// TIA Portal V20 export
FUNCTION_BLOCK "Sequence_1_Conveyor"   // FB157, LAD
TITLE = Sequence
// Sequence template programmend in ladder logic
// stored: IsIECCheckEnabled true, MemoryReserve 100, Namespace Unit1.Em7, SetENOAutomatically true
   VAR_INPUT
      UnitStatus : "LAF_typeUnitStatus";
   END_VAR
   VAR_OUTPUT
      safeState : Bool;
   END_VAR
   VAR
      instSequenceLADControl { ExternalWritable := 'False'} : "LAF_ControlLadSequence";
      instSequenceLADStatus { ExternalWritable := 'False'} : "LAF_StatusLadSequence";
      statPulse { ExternalWritable := 'False'} : Array[0..999] of Bool;
      statTonTimer { ExternalWritable := 'False'} : Array[0..1999] of TON_TIME;
   END_VAR
   VAR_TEMP
      tempCustomerAction : Bool;   // Placeholder for possible actions
      tempDo_nothing_and_wait_for_init : Bool;   // Placeholder for doing nothing
      tempSafeStateCondition : Bool;   // Temp Condition for the equipment module to be in a safe state
   END_VAR
   VAR CONSTANT
      STEP_IDLE : DInt := 1;   // Idle Step
      JOB_1_STEP_01 : DInt := 101;
      JOB_1_STEP_11 : DInt := 111;
      JOB_1_STEP_21 : DInt := 121;
      JOB_1_STEP_31 : DInt := 131;
      JOB_1_STEP_41 : DInt := 141;
      JOB_1_STEP_51 : DInt := 151;
      JOB_1_STEP_61 : DInt := 161;
      JOB_1_STEP_71 : DInt := 171;
      JOB_1_STEP_81 : DInt := 181;
      JOB_1_STEP_91 : DInt := 191;
      JOB_2_STEP_01 : DInt := 201;
      JOB_2_STEP_11 : DInt := 211;
      JOB_2_STEP_21 : DInt := 221;
      JOB_2_STEP_31 : DInt := 231;
      JOB_2_STEP_41 : DInt := 241;
      JOB_2_STEP_51 : DInt := 251;
      JOB_2_STEP_61 : DInt := 261;
      JOB_2_STEP_71 : DInt := 271;
      JOB_2_STEP_81 : DInt := 281;
      JOB_2_STEP_91 : DInt := 291;
      JOB_3_STEP_01 : DInt := 301;
      JOB_3_STEP_11 : DInt := 311;
      JOB_3_STEP_21 : DInt := 321;
      JOB_3_STEP_31 : DInt := 331;
      JOB_3_STEP_41 : DInt := 341;
      JOB_3_STEP_51 : DInt := 351;
      JOB_3_STEP_61 : DInt := 361;
      JOB_3_STEP_71 : DInt := 371;
      JOB_3_STEP_81 : DInt := 381;
      JOB_3_STEP_91 : DInt := 391;
      JOB_4_STEP_01 : DInt := 401;
      JOB_4_STEP_11 : DInt := 411;
      JOB_4_STEP_21 : DInt := 421;
      JOB_4_STEP_31 : DInt := 431;
      JOB_4_STEP_41 : DInt := 441;
      JOB_4_STEP_51 : DInt := 451;
      JOB_4_STEP_61 : DInt := 461;
      JOB_4_STEP_71 : DInt := 471;
      JOB_4_STEP_81 : DInt := 481;
      JOB_4_STEP_91 : DInt := 491;
      JOB_8_STEP_01 : DInt := 801;
      JOB_8_STEP_11 : DInt := 811;
      JOB_8_STEP_21 : DInt := 821;
      JOB_8_STEP_31 : DInt := 831;
      JOB_8_STEP_41 : DInt := 841;
      JOB_8_STEP_51 : DInt := 851;
      JOB_8_STEP_61 : DInt := 861;
      JOB_8_STEP_71 : DInt := 871;
      JOB_8_STEP_81 : DInt := 881;
      JOB_8_STEP_91 : DInt := 891;
      JOB_9_STEP_01 : DInt := 901;
      JOB_9_STEP_11 : DInt := 911;
      JOB_9_STEP_21 : DInt := 921;
      JOB_9_STEP_31 : DInt := 931;
      JOB_9_STEP_41 : DInt := 941;
      JOB_9_STEP_51 : DInt := 951;
      JOB_9_STEP_61 : DInt := 961;
      JOB_9_STEP_71 : DInt := 971;
      JOB_9_STEP_81 : DInt := 981;
      JOB_9_STEP_91 : DInt := 991;
      JOB_10_STEP_01 : DInt := 1001;
      JOB_10_STEP_11 : DInt := 1011;
      JOB_10_STEP_21 : DInt := 1021;
      JOB_10_STEP_31 : DInt := 1031;
      JOB_10_STEP_41 : DInt := 1041;
      JOB_10_STEP_51 : DInt := 1051;
      JOB_10_STEP_61 : DInt := 1061;
      JOB_10_STEP_71 : DInt := 1071;
      JOB_10_STEP_81 : DInt := 1081;
      JOB_10_STEP_91 : DInt := 1091;
      JOB_11_STEP_01 : DInt := 1101;
      JOB_11_STEP_11 : DInt := 1111;
      JOB_11_STEP_21 : DInt := 1121;
      JOB_11_STEP_31 : DInt := 1131;
      JOB_11_STEP_41 : DInt := 1141;
      JOB_11_STEP_51 : DInt := 1151;
      JOB_11_STEP_61 : DInt := 1161;
      JOB_11_STEP_71 : DInt := 1171;
      JOB_11_STEP_81 : DInt := 1181;
      JOB_11_STEP_91 : DInt := 1191;
      JOB_12_STEP_01 : DInt := 1201;
      JOB_12_STEP_11 : DInt := 1211;
      JOB_12_STEP_21 : DInt := 1221;
      JOB_12_STEP_31 : DInt := 1231;
      JOB_12_STEP_41 : DInt := 1241;
      JOB_12_STEP_51 : DInt := 1251;
      JOB_12_STEP_61 : DInt := 1261;
      JOB_12_STEP_71 : DInt := 1271;
      JOB_12_STEP_81 : DInt := 1281;
      JOB_12_STEP_91 : DInt := 1291;
      STEP_IMMEDIATE_STOP : DInt := 9001;   // Step executed when an immediate stop command is triggered for the sequence (i.e. when unit is in state aborting)
      SeqDelayTime : Time := T#100ms;
      SeqNoDelayTime : Time;
      TRUE : Bool := TRUE;
      FALSE : Bool := FALSE;
      All_CV_Move : DInt := 1103;
      Stack2_Not_Move : DInt := 1105;
      Stack1_Work : DInt := 1110;
      Stack2_Work : DInt := 1115;
      Stack_Full_Check : DInt := 1120;
      "2Pitch_Move" : DInt := 1130;
      "Stack1+Stack2_Work" : DInt := 1140;
   END_VAR
   VAR_TEMP   // added for the SCL form of the ladder/FBD networks
      _w1 : Bool;
      _w2 : Bool;
      _w3 : Bool;
   END_VAR
BEGIN

REGION Network 1: BLOCK INFO HEADER
   // (company) / (C) Copyright (year)
   // ---------------------------------------------------------------------------------
   // Title:                             (Title of this block)
   // Comment/Function: (that is implemented in the block)
   // Library/Family:           (that the source is dedicated to)
   // Author:                        (department / person in charge / contact)
   // Target System:          (test system with FW version)
   // Engineering:              TIA Portal (SW version)
   // Restrictions:               (OB types, etc.)
   // Requirements:           (hardware, technological package, etc.)
   // ---------------------------------------------------------------------------------
   // Change log table:
   // Version          | Date             | Signature      | Expert in charge  | Changes applied ------------------------|----------------------|-------------------------|--------------------------------|-----------------------
   // 001.000.000 | yyyy-mm-dd | 0x00000000 | (name of expert) | First released version
END_REGION

REGION Network 2: DESCRIPTION
   // This is a template block provided by the Automation Framework. It can be used to create an own project.
   // The Block Info Header is prepared to put in your own data.
   // Description of the block could be added here and the docu created by Code2Docu.
END_REGION

REGION Network 3: *************** CONTROL **********************
END_REGION

REGION Network 4: Sequence Control
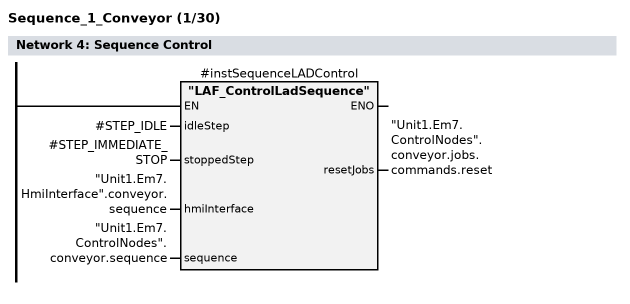
   RUNG wire#powerrail
      #instSequenceLADControl(idleStep := #STEP_IDLE, stoppedStep := #STEP_IMMEDIATE_STOP, hmiInterface := "Unit1.Em7.HmiInterface".conveyor.sequence, sequence := "Unit1.Em7.ControlNodes".conveyor.sequence, resetJobs => "Unit1.Em7.ControlNodes".conveyor.jobs.commands.reset)
   END_RUNG
   // the same network as SCL:
   #instSequenceLADControl(idleStep := #STEP_IDLE,   // "LAF_ControlLadSequence"
                           stoppedStep := #STEP_IMMEDIATE_STOP,
                           hmiInterface := "Unit1.Em7.HmiInterface".conveyor.sequence,
                           sequence := "Unit1.Em7.ControlNodes".conveyor.sequence,
                           resetJobs => "Unit1.Em7.ControlNodes".conveyor.jobs.commands.reset);
END_REGION

REGION Network 5: Step IDLE
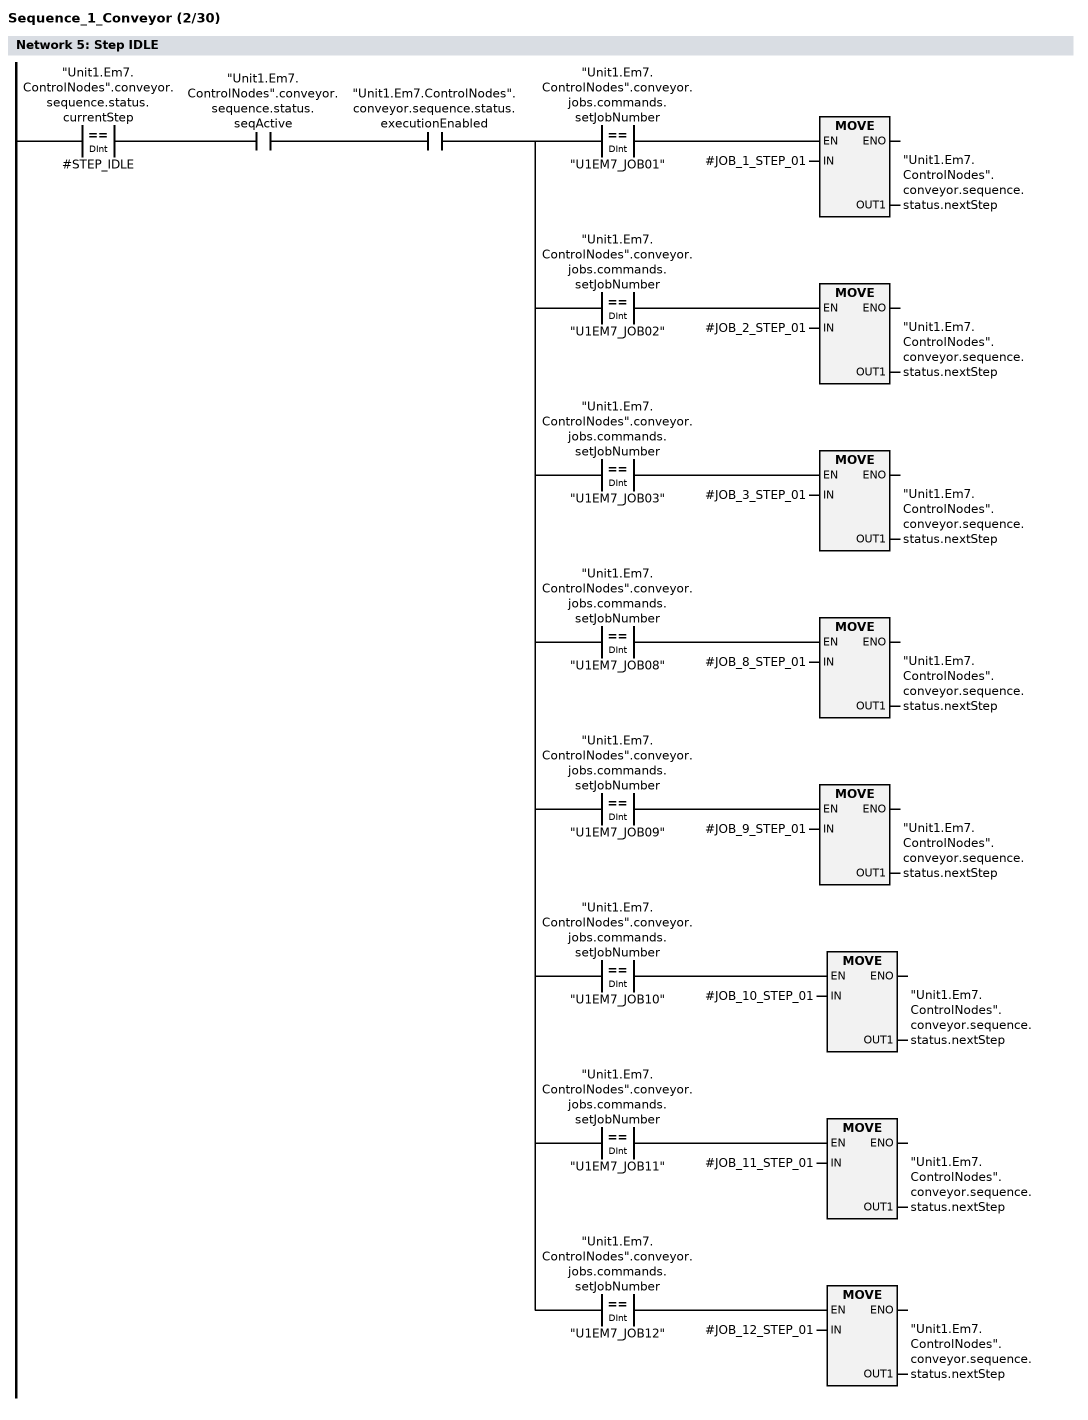
   RUNG wire#powerrail
      { S7_Templates := "SrcType := DInt" } EQ_Contact(in1 := "Unit1.Em7.ControlNodes".conveyor.sequence.status.currentStep, in2 := #STEP_IDLE)
      Contact( "Unit1.Em7.ControlNodes".conveyor.sequence.status.seqActive )
      Contact( "Unit1.Em7.ControlNodes".conveyor.sequence.status.executionEnabled )
      wire#w1
      { S7_Templates := "SrcType := DInt" } EQ_Contact(in1 := "Unit1.Em7.ControlNodes".conveyor.jobs.commands.setJobNumber, in2 := "U1EM7_JOB01")
      Move(in := #JOB_1_STEP_01, out1 => "Unit1.Em7.ControlNodes".conveyor.sequence.status.nextStep)
   END_RUNG
   RUNG wire#w1
      { S7_Templates := "SrcType := DInt" } EQ_Contact(in1 := "Unit1.Em7.ControlNodes".conveyor.jobs.commands.setJobNumber, in2 := "U1EM7_JOB02")
      Move(in := #JOB_2_STEP_01, out1 => "Unit1.Em7.ControlNodes".conveyor.sequence.status.nextStep)
   END_RUNG
   RUNG wire#w1
      { S7_Templates := "SrcType := DInt" } EQ_Contact(in1 := "Unit1.Em7.ControlNodes".conveyor.jobs.commands.setJobNumber, in2 := "U1EM7_JOB03")
      Move(in := #JOB_3_STEP_01, out1 => "Unit1.Em7.ControlNodes".conveyor.sequence.status.nextStep)
   END_RUNG
   RUNG wire#w1
      { S7_Templates := "SrcType := DInt" } EQ_Contact(in1 := "Unit1.Em7.ControlNodes".conveyor.jobs.commands.setJobNumber, in2 := "U1EM7_JOB08")
      Move(in := #JOB_8_STEP_01, out1 => "Unit1.Em7.ControlNodes".conveyor.sequence.status.nextStep)
   END_RUNG
   RUNG wire#w1
      { S7_Templates := "SrcType := DInt" } EQ_Contact(in1 := "Unit1.Em7.ControlNodes".conveyor.jobs.commands.setJobNumber, in2 := "U1EM7_JOB09")
      Move(in := #JOB_9_STEP_01, out1 => "Unit1.Em7.ControlNodes".conveyor.sequence.status.nextStep)
   END_RUNG
   RUNG wire#w1
      { S7_Templates := "SrcType := DInt" } EQ_Contact(in1 := "Unit1.Em7.ControlNodes".conveyor.jobs.commands.setJobNumber, in2 := "U1EM7_JOB10")
      Move(in := #JOB_10_STEP_01, out1 => "Unit1.Em7.ControlNodes".conveyor.sequence.status.nextStep)
   END_RUNG
   RUNG wire#w1
      { S7_Templates := "SrcType := DInt" } EQ_Contact(in1 := "Unit1.Em7.ControlNodes".conveyor.jobs.commands.setJobNumber, in2 := "U1EM7_JOB11")
      Move(in := #JOB_11_STEP_01, out1 => "Unit1.Em7.ControlNodes".conveyor.sequence.status.nextStep)
   END_RUNG
   RUNG wire#w1
      { S7_Templates := "SrcType := DInt" } EQ_Contact(in1 := "Unit1.Em7.ControlNodes".conveyor.jobs.commands.setJobNumber, in2 := "U1EM7_JOB12")
      Move(in := #JOB_12_STEP_01, out1 => "Unit1.Em7.ControlNodes".conveyor.sequence.status.nextStep)
   END_RUNG
   // the same network as SCL:
   #_w1 := ("Unit1.Em7.ControlNodes".conveyor.sequence.status.currentStep = #STEP_IDLE) AND "Unit1.Em7.ControlNodes".conveyor.sequence.status.seqActive AND "Unit1.Em7.ControlNodes".conveyor.sequence.status.executionEnabled;
   IF #_w1 AND ("Unit1.Em7.ControlNodes".conveyor.jobs.commands.setJobNumber = "U1EM7_JOB01") THEN
       "Unit1.Em7.ControlNodes".conveyor.sequence.status.nextStep := #JOB_1_STEP_01;
   END_IF;
   IF #_w1 AND ("Unit1.Em7.ControlNodes".conveyor.jobs.commands.setJobNumber = "U1EM7_JOB02") THEN
       "Unit1.Em7.ControlNodes".conveyor.sequence.status.nextStep := #JOB_2_STEP_01;
   END_IF;
   IF #_w1 AND ("Unit1.Em7.ControlNodes".conveyor.jobs.commands.setJobNumber = "U1EM7_JOB03") THEN
       "Unit1.Em7.ControlNodes".conveyor.sequence.status.nextStep := #JOB_3_STEP_01;
   END_IF;
   IF #_w1 AND ("Unit1.Em7.ControlNodes".conveyor.jobs.commands.setJobNumber = "U1EM7_JOB08") THEN
       "Unit1.Em7.ControlNodes".conveyor.sequence.status.nextStep := #JOB_8_STEP_01;
   END_IF;
   IF #_w1 AND ("Unit1.Em7.ControlNodes".conveyor.jobs.commands.setJobNumber = "U1EM7_JOB09") THEN
       "Unit1.Em7.ControlNodes".conveyor.sequence.status.nextStep := #JOB_9_STEP_01;
   END_IF;
   IF #_w1 AND ("Unit1.Em7.ControlNodes".conveyor.jobs.commands.setJobNumber = "U1EM7_JOB10") THEN
       "Unit1.Em7.ControlNodes".conveyor.sequence.status.nextStep := #JOB_10_STEP_01;
   END_IF;
   IF #_w1 AND ("Unit1.Em7.ControlNodes".conveyor.jobs.commands.setJobNumber = "U1EM7_JOB11") THEN
       "Unit1.Em7.ControlNodes".conveyor.sequence.status.nextStep := #JOB_11_STEP_01;
   END_IF;
   IF #_w1 AND ("Unit1.Em7.ControlNodes".conveyor.jobs.commands.setJobNumber = "U1EM7_JOB12") THEN
       "Unit1.Em7.ControlNodes".conveyor.sequence.status.nextStep := #JOB_12_STEP_01;
   END_IF;
END_REGION

REGION Network 6: ******************** JOB[1] EM INITIALIZED ********************
END_REGION

REGION Network 7: Step[101] : JOB[1] Condition
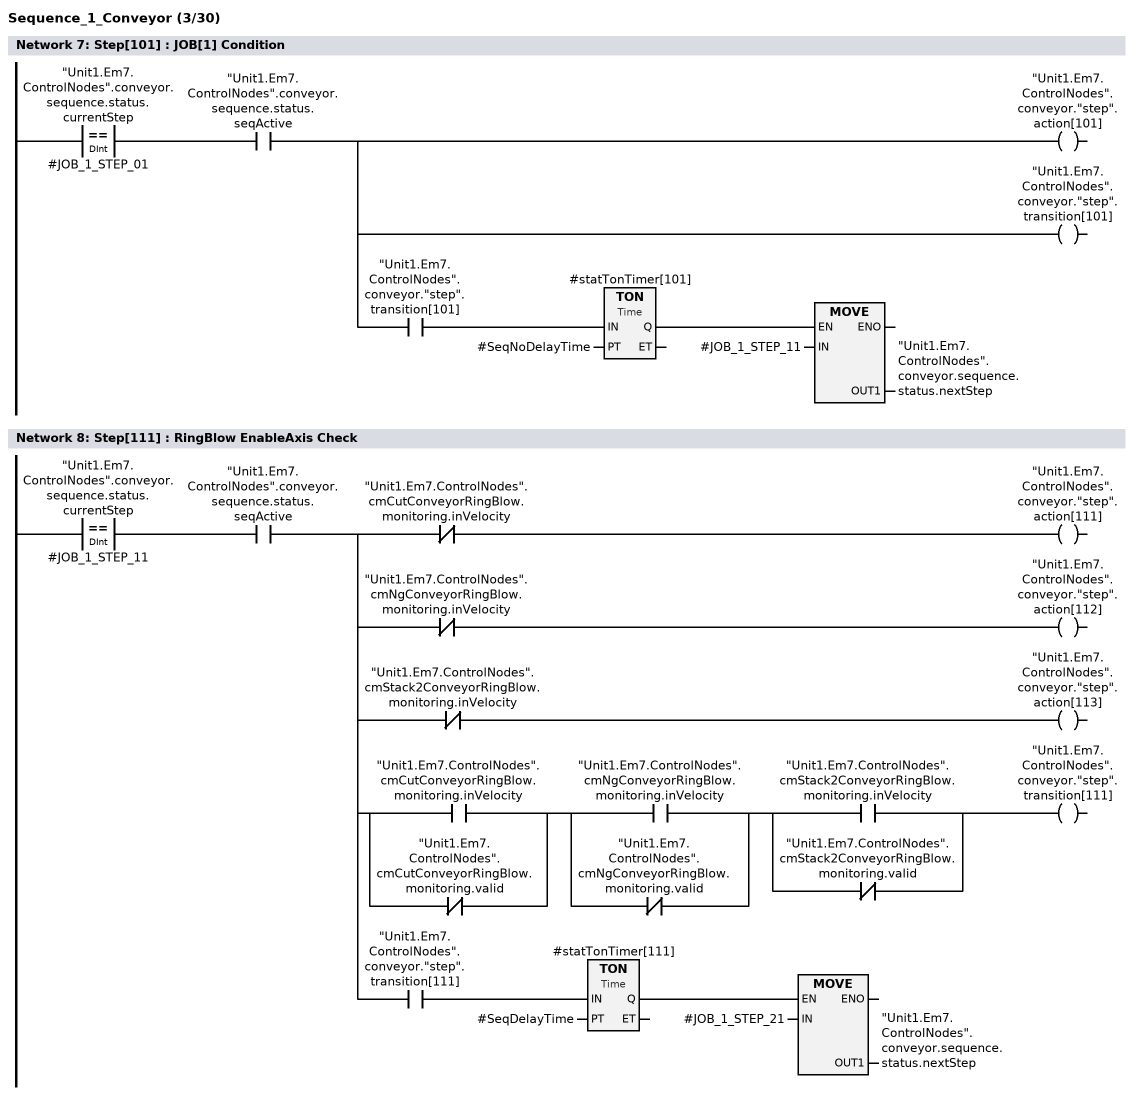
   RUNG wire#powerrail
      { S7_Templates := "SrcType := DInt" } EQ_Contact(in1 := "Unit1.Em7.ControlNodes".conveyor.sequence.status.currentStep, in2 := #JOB_1_STEP_01)
      Contact( "Unit1.Em7.ControlNodes".conveyor.sequence.status.seqActive )
      wire#w1
      Coil( "Unit1.Em7.ControlNodes".conveyor."step".action[101] )
   END_RUNG
   RUNG wire#w1
      Coil( "Unit1.Em7.ControlNodes".conveyor."step".transition[101] )
   END_RUNG
   RUNG wire#w1
      Contact( "Unit1.Em7.ControlNodes".conveyor."step".transition[101] )
      { S7_Templates := "time_type := Time" } #statTonTimer[101].TON(pt := #SeqNoDelayTime, et =>)
      Move(in := #JOB_1_STEP_11, out1 => "Unit1.Em7.ControlNodes".conveyor.sequence.status.nextStep)
   END_RUNG
   // the same network as SCL:
   "Unit1.Em7.ControlNodes".conveyor."step".action[101] := ("Unit1.Em7.ControlNodes".conveyor.sequence.status.currentStep = #JOB_1_STEP_01) AND "Unit1.Em7.ControlNodes".conveyor.sequence.status.seqActive;
   "Unit1.Em7.ControlNodes".conveyor."step".transition[101] := ("Unit1.Em7.ControlNodes".conveyor.sequence.status.currentStep = #JOB_1_STEP_01) AND "Unit1.Em7.ControlNodes".conveyor.sequence.status.seqActive;
   #statTonTimer[101].TON(IN := ("Unit1.Em7.ControlNodes".conveyor.sequence.status.currentStep = #JOB_1_STEP_01) AND "Unit1.Em7.ControlNodes".conveyor.sequence.status.seqActive AND "Unit1.Em7.ControlNodes".conveyor."step".transition[101],
                          PT := #SeqNoDelayTime);
   IF #statTonTimer[101].Q THEN
       "Unit1.Em7.ControlNodes".conveyor.sequence.status.nextStep := #JOB_1_STEP_11;
   END_IF;
END_REGION

REGION Network 8: Step[111] : RingBlow EnableAxis Check
   RUNG wire#powerrail
      { S7_Templates := "SrcType := DInt" } EQ_Contact(in1 := "Unit1.Em7.ControlNodes".conveyor.sequence.status.currentStep, in2 := #JOB_1_STEP_11)
      Contact( "Unit1.Em7.ControlNodes".conveyor.sequence.status.seqActive )
      wire#w1
      I_Contact( "Unit1.Em7.ControlNodes".cmCutConveyorRingBlow.monitoring.inVelocity )
      Coil( "Unit1.Em7.ControlNodes".conveyor."step".action[111] )
   END_RUNG
   RUNG wire#w1
      I_Contact( "Unit1.Em7.ControlNodes".cmNgConveyorRingBlow.monitoring.inVelocity )
      Coil( "Unit1.Em7.ControlNodes".conveyor."step".action[112] )
   END_RUNG
   RUNG wire#w1
      I_Contact( "Unit1.Em7.ControlNodes".cmStack2ConveyorRingBlow.monitoring.inVelocity )
      Coil( "Unit1.Em7.ControlNodes".conveyor."step".action[113] )
   END_RUNG
   RUNG wire#w1
      Contact( "Unit1.Em7.ControlNodes".cmCutConveyorRingBlow.monitoring.inVelocity )
      wire#w2
      Contact( "Unit1.Em7.ControlNodes".cmNgConveyorRingBlow.monitoring.inVelocity )
      wire#w3
      Contact( "Unit1.Em7.ControlNodes".cmStack2ConveyorRingBlow.monitoring.inVelocity )
      wire#w4
      Coil( "Unit1.Em7.ControlNodes".conveyor."step".transition[111] )
   END_RUNG
   RUNG wire#w1
      I_Contact( "Unit1.Em7.ControlNodes".cmCutConveyorRingBlow.monitoring.valid )
   END_RUNG wire#w2
   RUNG wire#w2
      I_Contact( "Unit1.Em7.ControlNodes".cmNgConveyorRingBlow.monitoring.valid )
   END_RUNG wire#w3
   RUNG wire#w3
      I_Contact( "Unit1.Em7.ControlNodes".cmStack2ConveyorRingBlow.monitoring.valid )
   END_RUNG wire#w4
   RUNG wire#w1
      Contact( "Unit1.Em7.ControlNodes".conveyor."step".transition[111] )
      { S7_Templates := "time_type := Time" } #statTonTimer[111].TON(pt := #SeqDelayTime, et =>)
      Move(in := #JOB_1_STEP_21, out1 => "Unit1.Em7.ControlNodes".conveyor.sequence.status.nextStep)
   END_RUNG
   // the same network as SCL:
   #_w1 := ("Unit1.Em7.ControlNodes".conveyor.sequence.status.currentStep = #JOB_1_STEP_11) AND "Unit1.Em7.ControlNodes".conveyor.sequence.status.seqActive;
   "Unit1.Em7.ControlNodes".conveyor."step".action[111] := #_w1 AND NOT "Unit1.Em7.ControlNodes".cmCutConveyorRingBlow.monitoring.inVelocity;
   "Unit1.Em7.ControlNodes".conveyor."step".action[112] := #_w1 AND NOT "Unit1.Em7.ControlNodes".cmNgConveyorRingBlow.monitoring.inVelocity;
   "Unit1.Em7.ControlNodes".conveyor."step".action[113] := #_w1 AND NOT "Unit1.Em7.ControlNodes".cmStack2ConveyorRingBlow.monitoring.inVelocity;
   "Unit1.Em7.ControlNodes".conveyor."step".transition[111] := #_w1 AND ("Unit1.Em7.ControlNodes".cmCutConveyorRingBlow.monitoring.inVelocity OR NOT "Unit1.Em7.ControlNodes".cmCutConveyorRingBlow.monitoring.valid) AND ("Unit1.Em7.ControlNodes".cmNgConveyorRingBlow.monitoring.inVelocity OR NOT "Unit1.Em7.ControlNodes".cmNgConveyorRingBlow.monitoring.valid) AND ("Unit1.Em7.ControlNodes".cmStack2ConveyorRingBlow.monitoring.inVelocity OR NOT "Unit1.Em7.ControlNodes".cmStack2ConveyorRingBlow.monitoring.valid);
   #statTonTimer[111].TON(IN := #_w1 AND "Unit1.Em7.ControlNodes".conveyor."step".transition[111],
                          PT := #SeqDelayTime);
   IF #statTonTimer[111].Q THEN
       "Unit1.Em7.ControlNodes".conveyor.sequence.status.nextStep := #JOB_1_STEP_21;
   END_IF;
END_REGION

REGION Network 9: Step[121] : Conveyor Axis B Homed Check
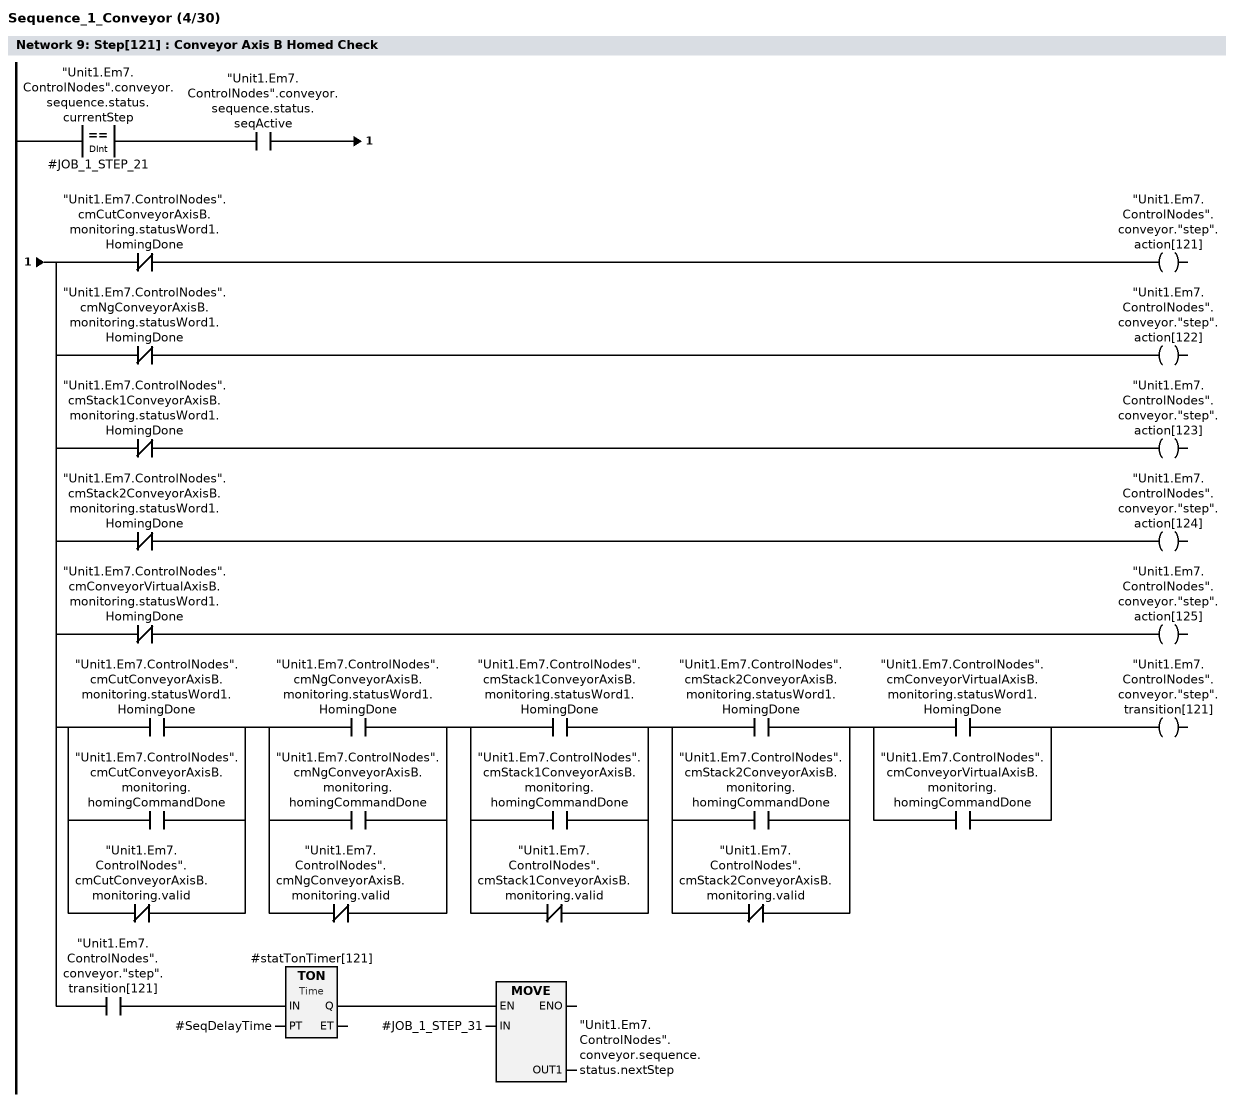
   RUNG wire#powerrail
      { S7_Templates := "SrcType := DInt" } EQ_Contact(in1 := "Unit1.Em7.ControlNodes".conveyor.sequence.status.currentStep, in2 := #JOB_1_STEP_21)
      Contact( "Unit1.Em7.ControlNodes".conveyor.sequence.status.seqActive )
      wire#w1
      I_Contact( "Unit1.Em7.ControlNodes".cmCutConveyorAxisB.monitoring.statusWord1.HomingDone )
      Coil( "Unit1.Em7.ControlNodes".conveyor."step".action[121] )
   END_RUNG
   RUNG wire#w1
      I_Contact( "Unit1.Em7.ControlNodes".cmNgConveyorAxisB.monitoring.statusWord1.HomingDone )
      Coil( "Unit1.Em7.ControlNodes".conveyor."step".action[122] )
   END_RUNG
   RUNG wire#w1
      I_Contact( "Unit1.Em7.ControlNodes".cmStack1ConveyorAxisB.monitoring.statusWord1.HomingDone )
      Coil( "Unit1.Em7.ControlNodes".conveyor."step".action[123] )
   END_RUNG
   RUNG wire#w1
      I_Contact( "Unit1.Em7.ControlNodes".cmStack2ConveyorAxisB.monitoring.statusWord1.HomingDone )
      Coil( "Unit1.Em7.ControlNodes".conveyor."step".action[124] )
   END_RUNG
   RUNG wire#w1
      I_Contact( "Unit1.Em7.ControlNodes".cmConveyorVirtualAxisB.monitoring.statusWord1.HomingDone )
      Coil( "Unit1.Em7.ControlNodes".conveyor."step".action[125] )
   END_RUNG
   RUNG wire#w1
      Contact( "Unit1.Em7.ControlNodes".cmCutConveyorAxisB.monitoring.statusWord1.HomingDone )
      wire#w2
      Contact( "Unit1.Em7.ControlNodes".cmNgConveyorAxisB.monitoring.statusWord1.HomingDone )
      wire#w3
      Contact( "Unit1.Em7.ControlNodes".cmStack1ConveyorAxisB.monitoring.statusWord1.HomingDone )
      wire#w4
      Contact( "Unit1.Em7.ControlNodes".cmStack2ConveyorAxisB.monitoring.statusWord1.HomingDone )
      wire#w5
      Contact( "Unit1.Em7.ControlNodes".cmConveyorVirtualAxisB.monitoring.statusWord1.HomingDone )
      wire#w6
      Coil( "Unit1.Em7.ControlNodes".conveyor."step".transition[121] )
   END_RUNG
   RUNG wire#w1
      Contact( "Unit1.Em7.ControlNodes".cmCutConveyorAxisB.monitoring.homingCommandDone )
   END_RUNG wire#w2
   RUNG wire#w1
      I_Contact( "Unit1.Em7.ControlNodes".cmCutConveyorAxisB.monitoring.valid )
   END_RUNG wire#w2
   RUNG wire#w2
      Contact( "Unit1.Em7.ControlNodes".cmNgConveyorAxisB.monitoring.homingCommandDone )
   END_RUNG wire#w3
   RUNG wire#w2
      I_Contact( "Unit1.Em7.ControlNodes".cmNgConveyorAxisB.monitoring.valid )
   END_RUNG wire#w3
   RUNG wire#w3
      Contact( "Unit1.Em7.ControlNodes".cmStack1ConveyorAxisB.monitoring.homingCommandDone )
   END_RUNG wire#w4
   RUNG wire#w3
      I_Contact( "Unit1.Em7.ControlNodes".cmStack1ConveyorAxisB.monitoring.valid )
   END_RUNG wire#w4
   RUNG wire#w4
      Contact( "Unit1.Em7.ControlNodes".cmStack2ConveyorAxisB.monitoring.homingCommandDone )
   END_RUNG wire#w5
   RUNG wire#w4
      I_Contact( "Unit1.Em7.ControlNodes".cmStack2ConveyorAxisB.monitoring.valid )
   END_RUNG wire#w5
   RUNG wire#w5
      Contact( "Unit1.Em7.ControlNodes".cmConveyorVirtualAxisB.monitoring.homingCommandDone )
   END_RUNG wire#w6
   RUNG wire#w1
      Contact( "Unit1.Em7.ControlNodes".conveyor."step".transition[121] )
      { S7_Templates := "time_type := Time" } #statTonTimer[121].TON(pt := #SeqDelayTime, et =>)
      Move(in := #JOB_1_STEP_31, out1 => "Unit1.Em7.ControlNodes".conveyor.sequence.status.nextStep)
   END_RUNG
   // the same network as SCL:
   #_w1 := ("Unit1.Em7.ControlNodes".conveyor.sequence.status.currentStep = #JOB_1_STEP_21) AND "Unit1.Em7.ControlNodes".conveyor.sequence.status.seqActive;
   "Unit1.Em7.ControlNodes".conveyor."step".action[121] := #_w1 AND NOT "Unit1.Em7.ControlNodes".cmCutConveyorAxisB.monitoring.statusWord1.HomingDone;
   "Unit1.Em7.ControlNodes".conveyor."step".action[122] := #_w1 AND NOT "Unit1.Em7.ControlNodes".cmNgConveyorAxisB.monitoring.statusWord1.HomingDone;
   "Unit1.Em7.ControlNodes".conveyor."step".action[123] := #_w1 AND NOT "Unit1.Em7.ControlNodes".cmStack1ConveyorAxisB.monitoring.statusWord1.HomingDone;
   "Unit1.Em7.ControlNodes".conveyor."step".action[124] := #_w1 AND NOT "Unit1.Em7.ControlNodes".cmStack2ConveyorAxisB.monitoring.statusWord1.HomingDone;
   "Unit1.Em7.ControlNodes".conveyor."step".action[125] := #_w1 AND NOT "Unit1.Em7.ControlNodes".cmConveyorVirtualAxisB.monitoring.statusWord1.HomingDone;
   "Unit1.Em7.ControlNodes".conveyor."step".transition[121] := #_w1 AND ("Unit1.Em7.ControlNodes".cmCutConveyorAxisB.monitoring.statusWord1.HomingDone OR "Unit1.Em7.ControlNodes".cmCutConveyorAxisB.monitoring.homingCommandDone OR NOT "Unit1.Em7.ControlNodes".cmCutConveyorAxisB.monitoring.valid) AND ("Unit1.Em7.ControlNodes".cmNgConveyorAxisB.monitoring.statusWord1.HomingDone OR "Unit1.Em7.ControlNodes".cmNgConveyorAxisB.monitoring.homingCommandDone OR NOT "Unit1.Em7.ControlNodes".cmNgConveyorAxisB.monitoring.valid) AND ("Unit1.Em7.ControlNodes".cmStack1ConveyorAxisB.monitoring.statusWord1.HomingDone OR "Unit1.Em7.ControlNodes".cmStack1ConveyorAxisB.monitoring.homingCommandDone OR NOT "Unit1.Em7.ControlNodes".cmStack1ConveyorAxisB.monitoring.valid) AND ("Unit1.Em7.ControlNodes".cmStack2ConveyorAxisB.monitoring.statusWord1.HomingDone OR "Unit1.Em7.ControlNodes".cmStack2ConveyorAxisB.monitoring.homingCommandDone OR NOT "Unit1.Em7.ControlNodes".cmStack2ConveyorAxisB.monitoring.valid) AND ("Unit1.Em7.ControlNodes".cmConveyorVirtualAxisB.monitoring.statusWord1.HomingDone OR "Unit1.Em7.ControlNodes".cmConveyorVirtualAxisB.monitoring.homingCommandDone);
   #statTonTimer[121].TON(IN := #_w1 AND "Unit1.Em7.ControlNodes".conveyor."step".transition[121],
                          PT := #SeqDelayTime);
   IF #statTonTimer[121].Q THEN
       "Unit1.Em7.ControlNodes".conveyor.sequence.status.nextStep := #JOB_1_STEP_31;
   END_IF;
END_REGION

REGION Network 10: Step[131] : Ng Box Lock Cylinder WorkPos Check
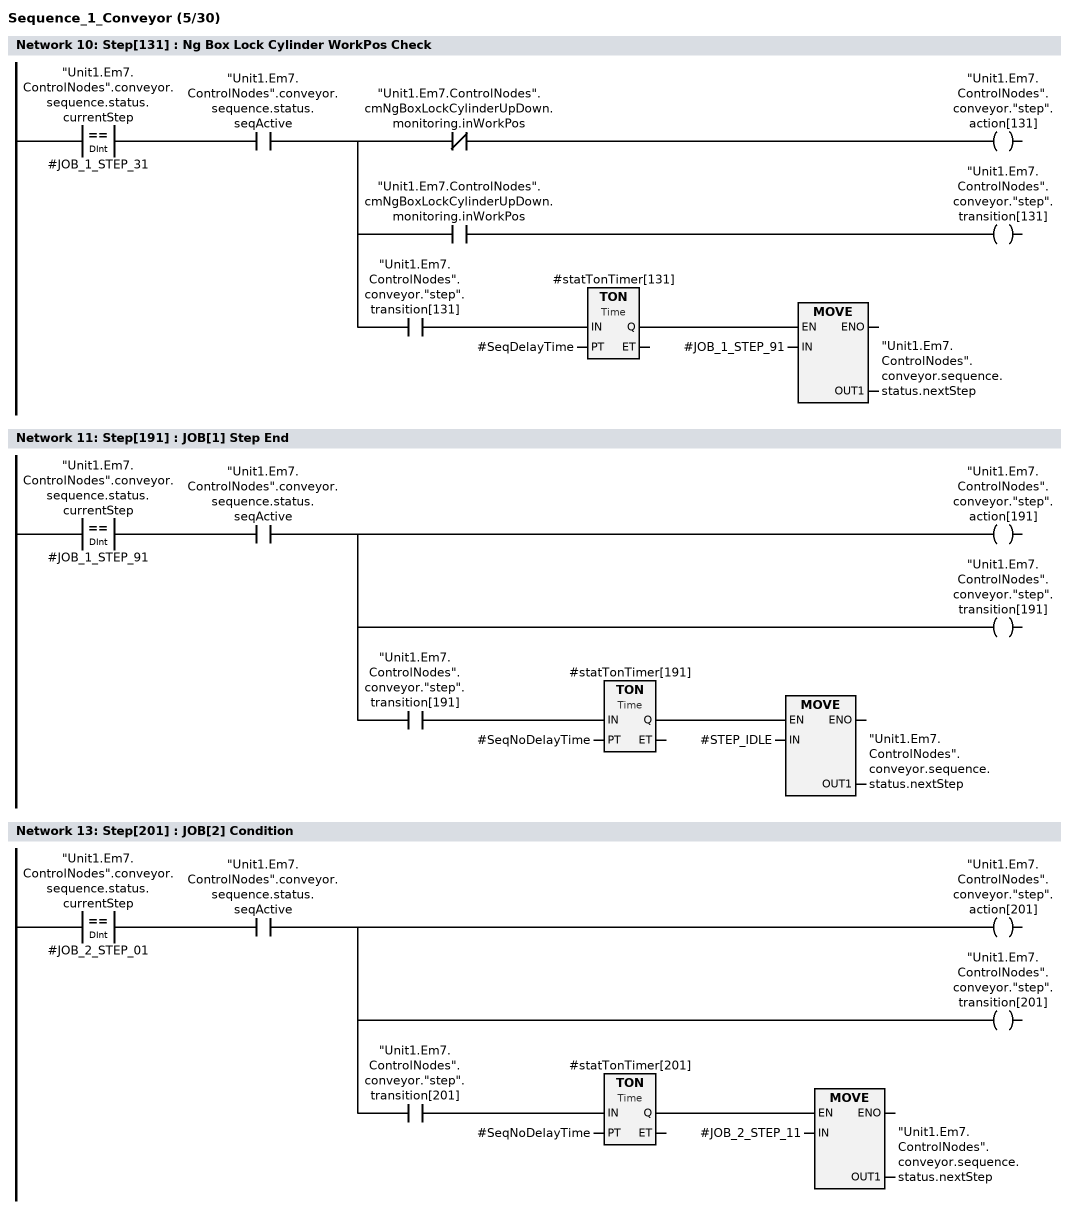
   RUNG wire#powerrail
      { S7_Templates := "SrcType := DInt" } EQ_Contact(in1 := "Unit1.Em7.ControlNodes".conveyor.sequence.status.currentStep, in2 := #JOB_1_STEP_31)
      Contact( "Unit1.Em7.ControlNodes".conveyor.sequence.status.seqActive )
      wire#w1
      I_Contact( "Unit1.Em7.ControlNodes".cmNgBoxLockCylinderUpDown.monitoring.inWorkPos )
      Coil( "Unit1.Em7.ControlNodes".conveyor."step".action[131] )
   END_RUNG
   RUNG wire#w1
      Contact( "Unit1.Em7.ControlNodes".cmNgBoxLockCylinderUpDown.monitoring.inWorkPos )
      Coil( "Unit1.Em7.ControlNodes".conveyor."step".transition[131] )
   END_RUNG
   RUNG wire#w1
      Contact( "Unit1.Em7.ControlNodes".conveyor."step".transition[131] )
      { S7_Templates := "time_type := Time" } #statTonTimer[131].TON(pt := #SeqDelayTime, et =>)
      Move(in := #JOB_1_STEP_91, out1 => "Unit1.Em7.ControlNodes".conveyor.sequence.status.nextStep)
   END_RUNG
   // the same network as SCL:
   #_w1 := ("Unit1.Em7.ControlNodes".conveyor.sequence.status.currentStep = #JOB_1_STEP_31) AND "Unit1.Em7.ControlNodes".conveyor.sequence.status.seqActive;
   "Unit1.Em7.ControlNodes".conveyor."step".action[131] := #_w1 AND NOT "Unit1.Em7.ControlNodes".cmNgBoxLockCylinderUpDown.monitoring.inWorkPos;
   "Unit1.Em7.ControlNodes".conveyor."step".transition[131] := #_w1 AND "Unit1.Em7.ControlNodes".cmNgBoxLockCylinderUpDown.monitoring.inWorkPos;
   #statTonTimer[131].TON(IN := #_w1 AND "Unit1.Em7.ControlNodes".conveyor."step".transition[131],
                          PT := #SeqDelayTime);
   IF #statTonTimer[131].Q THEN
       "Unit1.Em7.ControlNodes".conveyor.sequence.status.nextStep := #JOB_1_STEP_91;
   END_IF;
END_REGION

REGION Network 11: Step[191] : JOB[1] Step End
   RUNG wire#powerrail
      { S7_Templates := "SrcType := DInt" } EQ_Contact(in1 := "Unit1.Em7.ControlNodes".conveyor.sequence.status.currentStep, in2 := #JOB_1_STEP_91)
      Contact( "Unit1.Em7.ControlNodes".conveyor.sequence.status.seqActive )
      wire#w1
      Coil( "Unit1.Em7.ControlNodes".conveyor."step".action[191] )
   END_RUNG
   RUNG wire#w1
      Coil( "Unit1.Em7.ControlNodes".conveyor."step".transition[191] )
   END_RUNG
   RUNG wire#w1
      Contact( "Unit1.Em7.ControlNodes".conveyor."step".transition[191] )
      { S7_Templates := "time_type := Time" } #statTonTimer[191].TON(pt := #SeqNoDelayTime, et =>)
      Move(in := #STEP_IDLE, out1 => "Unit1.Em7.ControlNodes".conveyor.sequence.status.nextStep)
   END_RUNG
   // the same network as SCL:
   "Unit1.Em7.ControlNodes".conveyor."step".action[191] := ("Unit1.Em7.ControlNodes".conveyor.sequence.status.currentStep = #JOB_1_STEP_91) AND "Unit1.Em7.ControlNodes".conveyor.sequence.status.seqActive;
   "Unit1.Em7.ControlNodes".conveyor."step".transition[191] := ("Unit1.Em7.ControlNodes".conveyor.sequence.status.currentStep = #JOB_1_STEP_91) AND "Unit1.Em7.ControlNodes".conveyor.sequence.status.seqActive;
   #statTonTimer[191].TON(IN := ("Unit1.Em7.ControlNodes".conveyor.sequence.status.currentStep = #JOB_1_STEP_91) AND "Unit1.Em7.ControlNodes".conveyor.sequence.status.seqActive AND "Unit1.Em7.ControlNodes".conveyor."step".transition[191],
                          PT := #SeqNoDelayTime);
   IF #statTonTimer[191].Q THEN
       "Unit1.Em7.ControlNodes".conveyor.sequence.status.nextStep := #STEP_IDLE;
   END_IF;
END_REGION

REGION Network 12: ******************** JOB[2] CONVEYOR MOTION AUTO ********************
END_REGION

REGION Network 13: Step[201] : JOB[2] Condition
   RUNG wire#powerrail
      { S7_Templates := "SrcType := DInt" } EQ_Contact(in1 := "Unit1.Em7.ControlNodes".conveyor.sequence.status.currentStep, in2 := #JOB_2_STEP_01)
      Contact( "Unit1.Em7.ControlNodes".conveyor.sequence.status.seqActive )
      wire#w1
      Coil( "Unit1.Em7.ControlNodes".conveyor."step".action[201] )
   END_RUNG
   RUNG wire#w1
      Coil( "Unit1.Em7.ControlNodes".conveyor."step".transition[201] )
   END_RUNG
   RUNG wire#w1
      Contact( "Unit1.Em7.ControlNodes".conveyor."step".transition[201] )
      { S7_Templates := "time_type := Time" } #statTonTimer[201].TON(pt := #SeqNoDelayTime, et =>)
      Move(in := #JOB_2_STEP_11, out1 => "Unit1.Em7.ControlNodes".conveyor.sequence.status.nextStep)
   END_RUNG
   // the same network as SCL:
   "Unit1.Em7.ControlNodes".conveyor."step".action[201] := ("Unit1.Em7.ControlNodes".conveyor.sequence.status.currentStep = #JOB_2_STEP_01) AND "Unit1.Em7.ControlNodes".conveyor.sequence.status.seqActive;
   "Unit1.Em7.ControlNodes".conveyor."step".transition[201] := ("Unit1.Em7.ControlNodes".conveyor.sequence.status.currentStep = #JOB_2_STEP_01) AND "Unit1.Em7.ControlNodes".conveyor.sequence.status.seqActive;
   #statTonTimer[201].TON(IN := ("Unit1.Em7.ControlNodes".conveyor.sequence.status.currentStep = #JOB_2_STEP_01) AND "Unit1.Em7.ControlNodes".conveyor.sequence.status.seqActive AND "Unit1.Em7.ControlNodes".conveyor."step".transition[201],
                          PT := #SeqNoDelayTime);
   IF #statTonTimer[201].Q THEN
       "Unit1.Em7.ControlNodes".conveyor.sequence.status.nextStep := #JOB_2_STEP_11;
   END_IF;
END_REGION

REGION Network 14: Step[211] : Spare
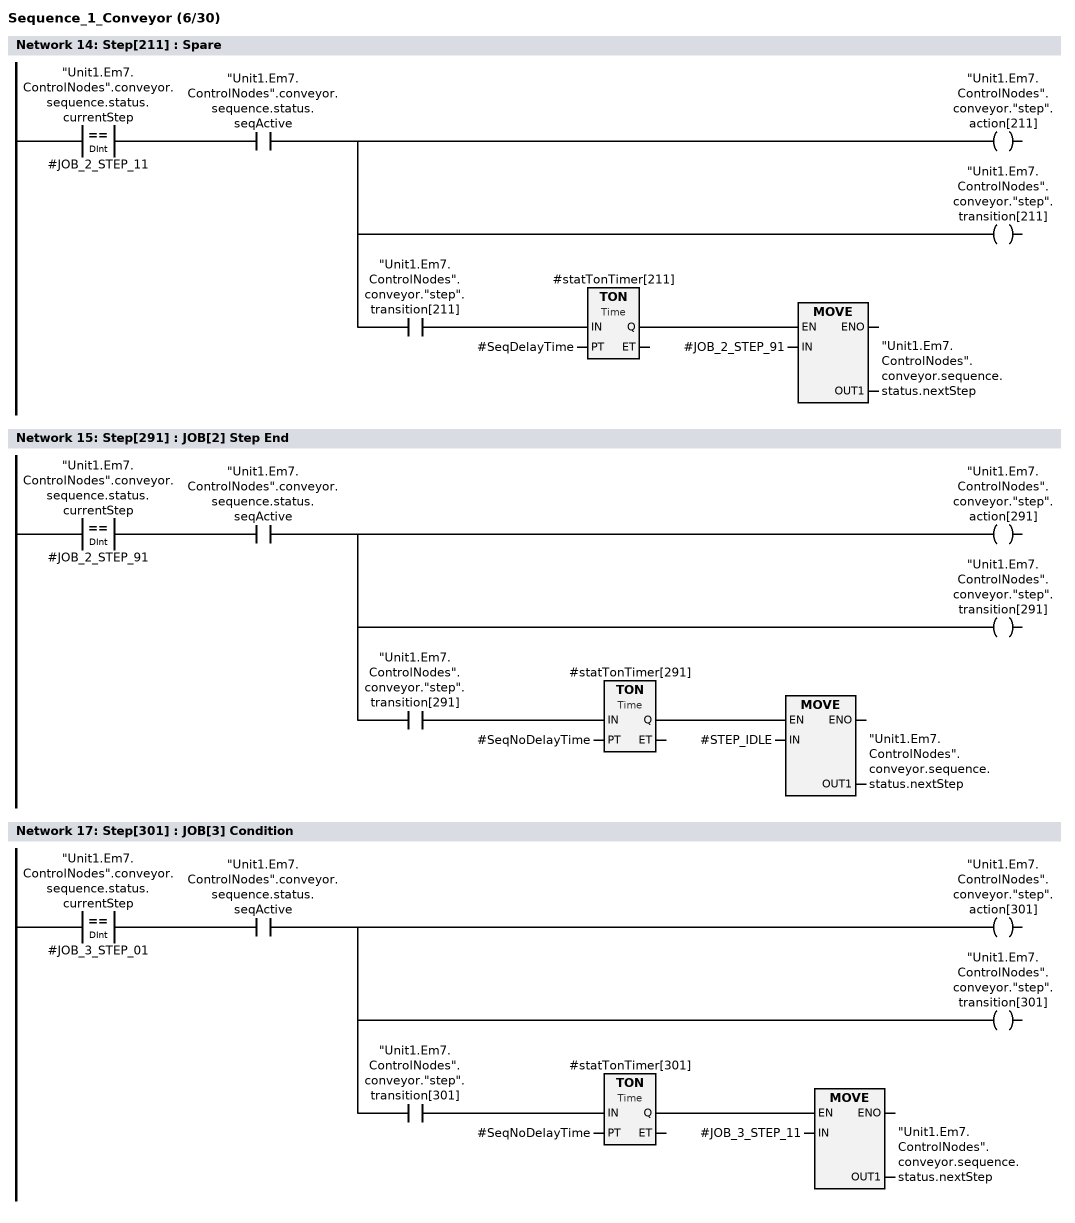
   RUNG wire#powerrail
      { S7_Templates := "SrcType := DInt" } EQ_Contact(in1 := "Unit1.Em7.ControlNodes".conveyor.sequence.status.currentStep, in2 := #JOB_2_STEP_11)
      Contact( "Unit1.Em7.ControlNodes".conveyor.sequence.status.seqActive )
      wire#w1
      Coil( "Unit1.Em7.ControlNodes".conveyor."step".action[211] )
   END_RUNG
   RUNG wire#w1
      Coil( "Unit1.Em7.ControlNodes".conveyor."step".transition[211] )
   END_RUNG
   RUNG wire#w1
      Contact( "Unit1.Em7.ControlNodes".conveyor."step".transition[211] )
      { S7_Templates := "time_type := Time" } #statTonTimer[211].TON(pt := #SeqDelayTime, et =>)
      Move(in := #JOB_2_STEP_91, out1 => "Unit1.Em7.ControlNodes".conveyor.sequence.status.nextStep)
   END_RUNG
   // the same network as SCL:
   "Unit1.Em7.ControlNodes".conveyor."step".action[211] := ("Unit1.Em7.ControlNodes".conveyor.sequence.status.currentStep = #JOB_2_STEP_11) AND "Unit1.Em7.ControlNodes".conveyor.sequence.status.seqActive;
   "Unit1.Em7.ControlNodes".conveyor."step".transition[211] := ("Unit1.Em7.ControlNodes".conveyor.sequence.status.currentStep = #JOB_2_STEP_11) AND "Unit1.Em7.ControlNodes".conveyor.sequence.status.seqActive;
   #statTonTimer[211].TON(IN := ("Unit1.Em7.ControlNodes".conveyor.sequence.status.currentStep = #JOB_2_STEP_11) AND "Unit1.Em7.ControlNodes".conveyor.sequence.status.seqActive AND "Unit1.Em7.ControlNodes".conveyor."step".transition[211],
                          PT := #SeqDelayTime);
   IF #statTonTimer[211].Q THEN
       "Unit1.Em7.ControlNodes".conveyor.sequence.status.nextStep := #JOB_2_STEP_91;
   END_IF;
END_REGION

REGION Network 15: Step[291] : JOB[2] Step End
   RUNG wire#powerrail
      { S7_Templates := "SrcType := DInt" } EQ_Contact(in1 := "Unit1.Em7.ControlNodes".conveyor.sequence.status.currentStep, in2 := #JOB_2_STEP_91)
      Contact( "Unit1.Em7.ControlNodes".conveyor.sequence.status.seqActive )
      wire#w1
      Coil( "Unit1.Em7.ControlNodes".conveyor."step".action[291] )
   END_RUNG
   RUNG wire#w1
      Coil( "Unit1.Em7.ControlNodes".conveyor."step".transition[291] )
   END_RUNG
   RUNG wire#w1
      Contact( "Unit1.Em7.ControlNodes".conveyor."step".transition[291] )
      { S7_Templates := "time_type := Time" } #statTonTimer[291].TON(pt := #SeqNoDelayTime, et =>)
      Move(in := #STEP_IDLE, out1 => "Unit1.Em7.ControlNodes".conveyor.sequence.status.nextStep)
   END_RUNG
   // the same network as SCL:
   "Unit1.Em7.ControlNodes".conveyor."step".action[291] := ("Unit1.Em7.ControlNodes".conveyor.sequence.status.currentStep = #JOB_2_STEP_91) AND "Unit1.Em7.ControlNodes".conveyor.sequence.status.seqActive;
   "Unit1.Em7.ControlNodes".conveyor."step".transition[291] := ("Unit1.Em7.ControlNodes".conveyor.sequence.status.currentStep = #JOB_2_STEP_91) AND "Unit1.Em7.ControlNodes".conveyor.sequence.status.seqActive;
   #statTonTimer[291].TON(IN := ("Unit1.Em7.ControlNodes".conveyor.sequence.status.currentStep = #JOB_2_STEP_91) AND "Unit1.Em7.ControlNodes".conveyor.sequence.status.seqActive AND "Unit1.Em7.ControlNodes".conveyor."step".transition[291],
                          PT := #SeqNoDelayTime);
   IF #statTonTimer[291].Q THEN
       "Unit1.Em7.ControlNodes".conveyor.sequence.status.nextStep := #STEP_IDLE;
   END_IF;
END_REGION

REGION Network 16: ******************** JOB[3] CONVEYOR PITCH AUTO ********************
END_REGION

REGION Network 17: Step[301] : JOB[3] Condition
   RUNG wire#powerrail
      { S7_Templates := "SrcType := DInt" } EQ_Contact(in1 := "Unit1.Em7.ControlNodes".conveyor.sequence.status.currentStep, in2 := #JOB_3_STEP_01)
      Contact( "Unit1.Em7.ControlNodes".conveyor.sequence.status.seqActive )
      wire#w1
      Coil( "Unit1.Em7.ControlNodes".conveyor."step".action[301] )
   END_RUNG
   RUNG wire#w1
      Coil( "Unit1.Em7.ControlNodes".conveyor."step".transition[301] )
   END_RUNG
   RUNG wire#w1
      Contact( "Unit1.Em7.ControlNodes".conveyor."step".transition[301] )
      { S7_Templates := "time_type := Time" } #statTonTimer[301].TON(pt := #SeqNoDelayTime, et =>)
      Move(in := #JOB_3_STEP_11, out1 => "Unit1.Em7.ControlNodes".conveyor.sequence.status.nextStep)
   END_RUNG
   // the same network as SCL:
   "Unit1.Em7.ControlNodes".conveyor."step".action[301] := ("Unit1.Em7.ControlNodes".conveyor.sequence.status.currentStep = #JOB_3_STEP_01) AND "Unit1.Em7.ControlNodes".conveyor.sequence.status.seqActive;
   "Unit1.Em7.ControlNodes".conveyor."step".transition[301] := ("Unit1.Em7.ControlNodes".conveyor.sequence.status.currentStep = #JOB_3_STEP_01) AND "Unit1.Em7.ControlNodes".conveyor.sequence.status.seqActive;
   #statTonTimer[301].TON(IN := ("Unit1.Em7.ControlNodes".conveyor.sequence.status.currentStep = #JOB_3_STEP_01) AND "Unit1.Em7.ControlNodes".conveyor.sequence.status.seqActive AND "Unit1.Em7.ControlNodes".conveyor."step".transition[301],
                          PT := #SeqNoDelayTime);
   IF #statTonTimer[301].Q THEN
       "Unit1.Em7.ControlNodes".conveyor.sequence.status.nextStep := #JOB_3_STEP_11;
   END_IF;
END_REGION

REGION Network 18: Step[311] : Conveyor GearIn Command
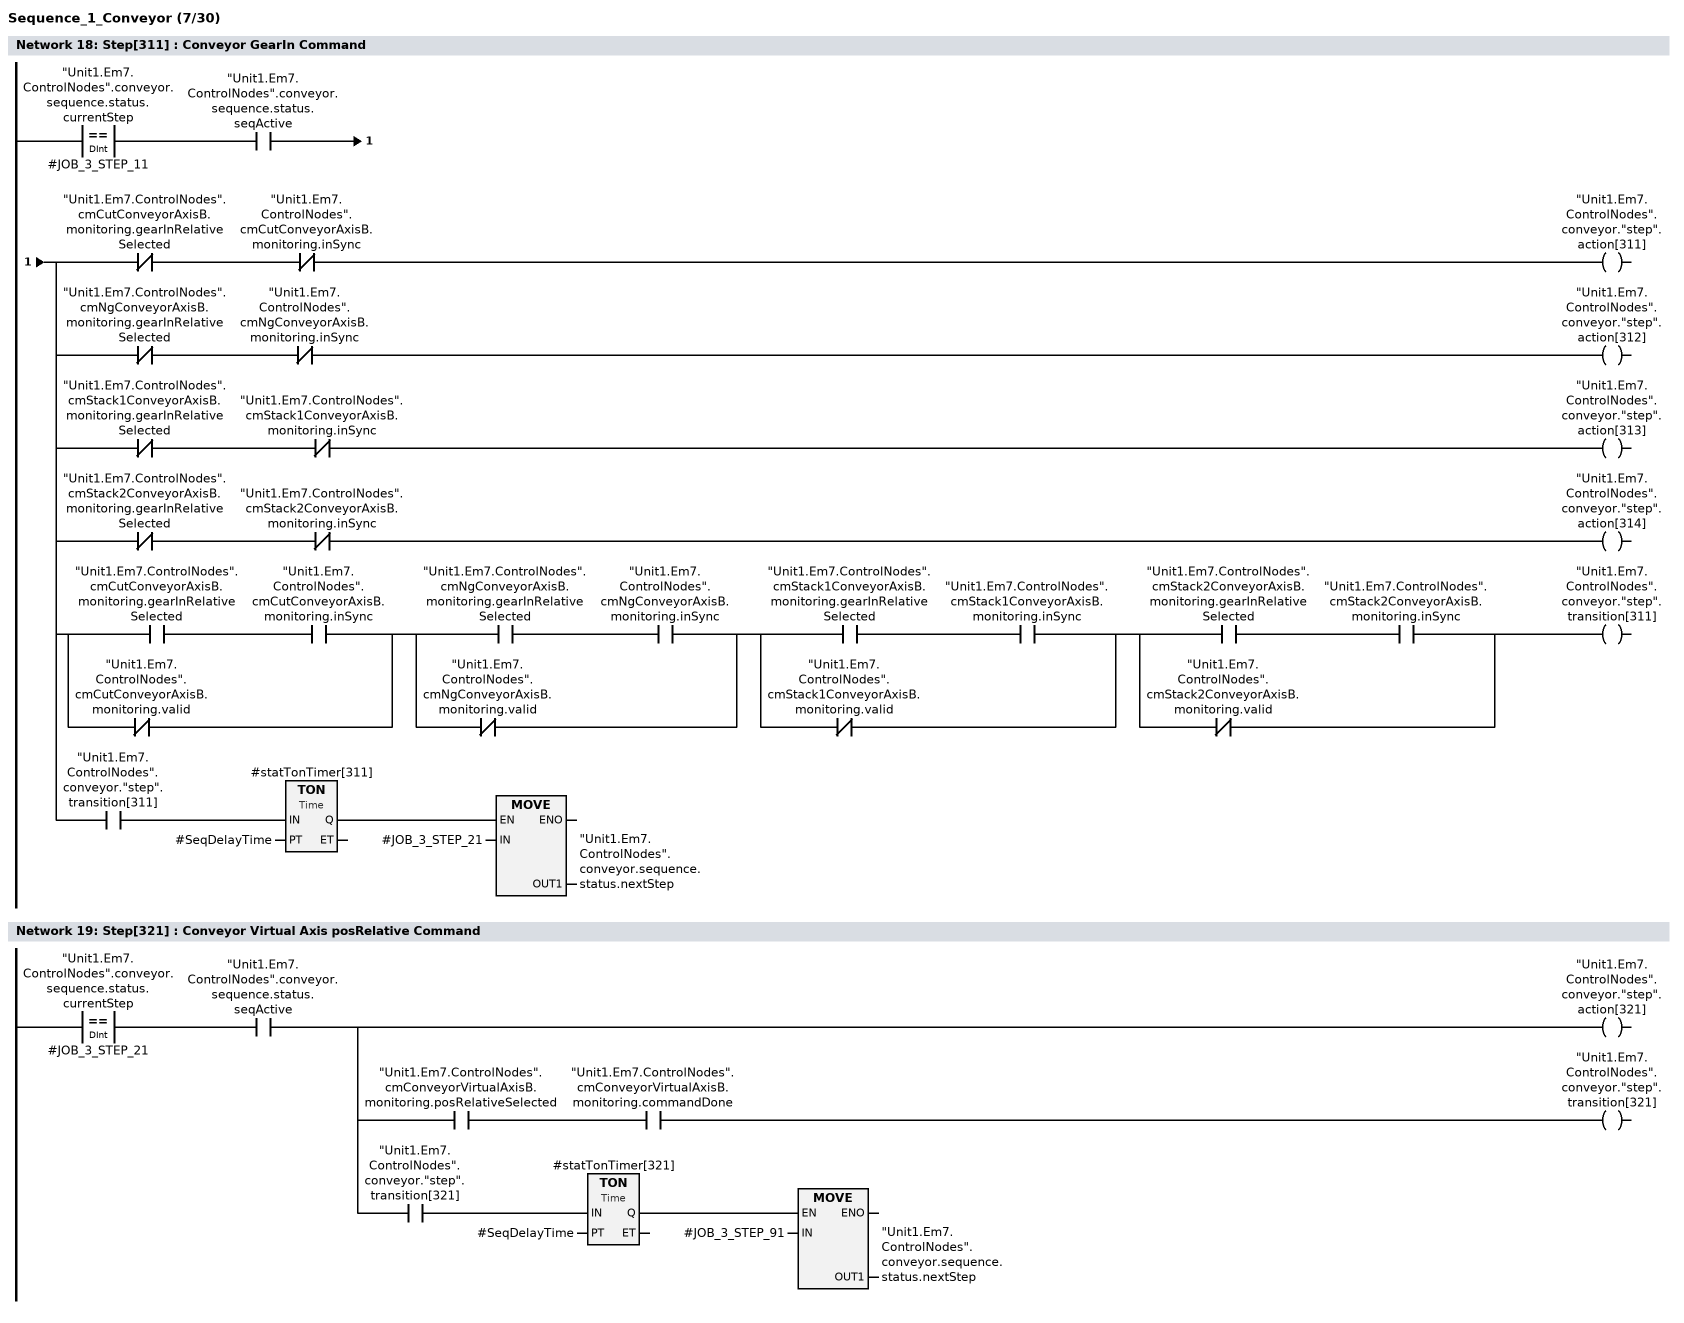
   RUNG wire#powerrail
      { S7_Templates := "SrcType := DInt" } EQ_Contact(in1 := "Unit1.Em7.ControlNodes".conveyor.sequence.status.currentStep, in2 := #JOB_3_STEP_11)
      Contact( "Unit1.Em7.ControlNodes".conveyor.sequence.status.seqActive )
      wire#w1
      I_Contact( "Unit1.Em7.ControlNodes".cmCutConveyorAxisB.monitoring.gearInRelativeSelected )
      I_Contact( "Unit1.Em7.ControlNodes".cmCutConveyorAxisB.monitoring.inSync )
      Coil( "Unit1.Em7.ControlNodes".conveyor."step".action[311] )
   END_RUNG
   RUNG wire#w1
      I_Contact( "Unit1.Em7.ControlNodes".cmNgConveyorAxisB.monitoring.gearInRelativeSelected )
      I_Contact( "Unit1.Em7.ControlNodes".cmNgConveyorAxisB.monitoring.inSync )
      Coil( "Unit1.Em7.ControlNodes".conveyor."step".action[312] )
   END_RUNG
   RUNG wire#w1
      I_Contact( "Unit1.Em7.ControlNodes".cmStack1ConveyorAxisB.monitoring.gearInRelativeSelected )
      I_Contact( "Unit1.Em7.ControlNodes".cmStack1ConveyorAxisB.monitoring.inSync )
      Coil( "Unit1.Em7.ControlNodes".conveyor."step".action[313] )
   END_RUNG
   RUNG wire#w1
      I_Contact( "Unit1.Em7.ControlNodes".cmStack2ConveyorAxisB.monitoring.gearInRelativeSelected )
      I_Contact( "Unit1.Em7.ControlNodes".cmStack2ConveyorAxisB.monitoring.inSync )
      Coil( "Unit1.Em7.ControlNodes".conveyor."step".action[314] )
   END_RUNG
   RUNG wire#w1
      Contact( "Unit1.Em7.ControlNodes".cmCutConveyorAxisB.monitoring.gearInRelativeSelected )
      Contact( "Unit1.Em7.ControlNodes".cmCutConveyorAxisB.monitoring.inSync )
      wire#w2
      Contact( "Unit1.Em7.ControlNodes".cmNgConveyorAxisB.monitoring.gearInRelativeSelected )
      Contact( "Unit1.Em7.ControlNodes".cmNgConveyorAxisB.monitoring.inSync )
      wire#w3
      Contact( "Unit1.Em7.ControlNodes".cmStack1ConveyorAxisB.monitoring.gearInRelativeSelected )
      Contact( "Unit1.Em7.ControlNodes".cmStack1ConveyorAxisB.monitoring.inSync )
      wire#w4
      Contact( "Unit1.Em7.ControlNodes".cmStack2ConveyorAxisB.monitoring.gearInRelativeSelected )
      Contact( "Unit1.Em7.ControlNodes".cmStack2ConveyorAxisB.monitoring.inSync )
      wire#w5
      Coil( "Unit1.Em7.ControlNodes".conveyor."step".transition[311] )
   END_RUNG
   RUNG wire#w1
      I_Contact( "Unit1.Em7.ControlNodes".cmCutConveyorAxisB.monitoring.valid )
   END_RUNG wire#w2
   RUNG wire#w2
      I_Contact( "Unit1.Em7.ControlNodes".cmNgConveyorAxisB.monitoring.valid )
   END_RUNG wire#w3
   RUNG wire#w3
      I_Contact( "Unit1.Em7.ControlNodes".cmStack1ConveyorAxisB.monitoring.valid )
   END_RUNG wire#w4
   RUNG wire#w4
      I_Contact( "Unit1.Em7.ControlNodes".cmStack2ConveyorAxisB.monitoring.valid )
   END_RUNG wire#w5
   RUNG wire#w1
      Contact( "Unit1.Em7.ControlNodes".conveyor."step".transition[311] )
      { S7_Templates := "time_type := Time" } #statTonTimer[311].TON(pt := #SeqDelayTime, et =>)
      Move(in := #JOB_3_STEP_21, out1 => "Unit1.Em7.ControlNodes".conveyor.sequence.status.nextStep)
   END_RUNG
   // the same network as SCL:
   #_w1 := ("Unit1.Em7.ControlNodes".conveyor.sequence.status.currentStep = #JOB_3_STEP_11) AND "Unit1.Em7.ControlNodes".conveyor.sequence.status.seqActive;
   "Unit1.Em7.ControlNodes".conveyor."step".action[311] := #_w1 AND NOT "Unit1.Em7.ControlNodes".cmCutConveyorAxisB.monitoring.gearInRelativeSelected AND NOT "Unit1.Em7.ControlNodes".cmCutConveyorAxisB.monitoring.inSync;
   "Unit1.Em7.ControlNodes".conveyor."step".action[312] := #_w1 AND NOT "Unit1.Em7.ControlNodes".cmNgConveyorAxisB.monitoring.gearInRelativeSelected AND NOT "Unit1.Em7.ControlNodes".cmNgConveyorAxisB.monitoring.inSync;
   "Unit1.Em7.ControlNodes".conveyor."step".action[313] := #_w1 AND NOT "Unit1.Em7.ControlNodes".cmStack1ConveyorAxisB.monitoring.gearInRelativeSelected AND NOT "Unit1.Em7.ControlNodes".cmStack1ConveyorAxisB.monitoring.inSync;
   "Unit1.Em7.ControlNodes".conveyor."step".action[314] := #_w1 AND NOT "Unit1.Em7.ControlNodes".cmStack2ConveyorAxisB.monitoring.gearInRelativeSelected AND NOT "Unit1.Em7.ControlNodes".cmStack2ConveyorAxisB.monitoring.inSync;
   "Unit1.Em7.ControlNodes".conveyor."step".transition[311] := #_w1 AND (("Unit1.Em7.ControlNodes".cmCutConveyorAxisB.monitoring.gearInRelativeSelected AND "Unit1.Em7.ControlNodes".cmCutConveyorAxisB.monitoring.inSync) OR NOT "Unit1.Em7.ControlNodes".cmCutConveyorAxisB.monitoring.valid) AND (("Unit1.Em7.ControlNodes".cmNgConveyorAxisB.monitoring.gearInRelativeSelected AND "Unit1.Em7.ControlNodes".cmNgConveyorAxisB.monitoring.inSync) OR NOT "Unit1.Em7.ControlNodes".cmNgConveyorAxisB.monitoring.valid) AND (("Unit1.Em7.ControlNodes".cmStack1ConveyorAxisB.monitoring.gearInRelativeSelected AND "Unit1.Em7.ControlNodes".cmStack1ConveyorAxisB.monitoring.inSync) OR NOT "Unit1.Em7.ControlNodes".cmStack1ConveyorAxisB.monitoring.valid) AND (("Unit1.Em7.ControlNodes".cmStack2ConveyorAxisB.monitoring.gearInRelativeSelected AND "Unit1.Em7.ControlNodes".cmStack2ConveyorAxisB.monitoring.inSync) OR NOT "Unit1.Em7.ControlNodes".cmStack2ConveyorAxisB.monitoring.valid);
   #statTonTimer[311].TON(IN := #_w1 AND "Unit1.Em7.ControlNodes".conveyor."step".transition[311],
                          PT := #SeqDelayTime);
   IF #statTonTimer[311].Q THEN
       "Unit1.Em7.ControlNodes".conveyor.sequence.status.nextStep := #JOB_3_STEP_21;
   END_IF;
END_REGION

REGION Network 19: Step[321] : Conveyor Virtual Axis posRelative Command
   RUNG wire#powerrail
      { S7_Templates := "SrcType := DInt" } EQ_Contact(in1 := "Unit1.Em7.ControlNodes".conveyor.sequence.status.currentStep, in2 := #JOB_3_STEP_21)
      Contact( "Unit1.Em7.ControlNodes".conveyor.sequence.status.seqActive )
      wire#w1
      Coil( "Unit1.Em7.ControlNodes".conveyor."step".action[321] )
   END_RUNG
   RUNG wire#w1
      Contact( "Unit1.Em7.ControlNodes".cmConveyorVirtualAxisB.monitoring.posRelativeSelected )
      Contact( "Unit1.Em7.ControlNodes".cmConveyorVirtualAxisB.monitoring.commandDone )
      Coil( "Unit1.Em7.ControlNodes".conveyor."step".transition[321] )
   END_RUNG
   RUNG wire#w1
      Contact( "Unit1.Em7.ControlNodes".conveyor."step".transition[321] )
      { S7_Templates := "time_type := Time" } #statTonTimer[321].TON(pt := #SeqDelayTime, et =>)
      Move(in := #JOB_3_STEP_91, out1 => "Unit1.Em7.ControlNodes".conveyor.sequence.status.nextStep)
   END_RUNG
   // the same network as SCL:
   "Unit1.Em7.ControlNodes".conveyor."step".action[321] := ("Unit1.Em7.ControlNodes".conveyor.sequence.status.currentStep = #JOB_3_STEP_21) AND "Unit1.Em7.ControlNodes".conveyor.sequence.status.seqActive;
   "Unit1.Em7.ControlNodes".conveyor."step".transition[321] := ("Unit1.Em7.ControlNodes".conveyor.sequence.status.currentStep = #JOB_3_STEP_21) AND "Unit1.Em7.ControlNodes".conveyor.sequence.status.seqActive AND "Unit1.Em7.ControlNodes".cmConveyorVirtualAxisB.monitoring.posRelativeSelected AND "Unit1.Em7.ControlNodes".cmConveyorVirtualAxisB.monitoring.commandDone;
   #statTonTimer[321].TON(IN := ("Unit1.Em7.ControlNodes".conveyor.sequence.status.currentStep = #JOB_3_STEP_21) AND "Unit1.Em7.ControlNodes".conveyor.sequence.status.seqActive AND "Unit1.Em7.ControlNodes".conveyor."step".transition[321],
                          PT := #SeqDelayTime);
   IF #statTonTimer[321].Q THEN
       "Unit1.Em7.ControlNodes".conveyor.sequence.status.nextStep := #JOB_3_STEP_91;
   END_IF;
END_REGION

REGION Network 20: Step[391] : JOB[3] Step End
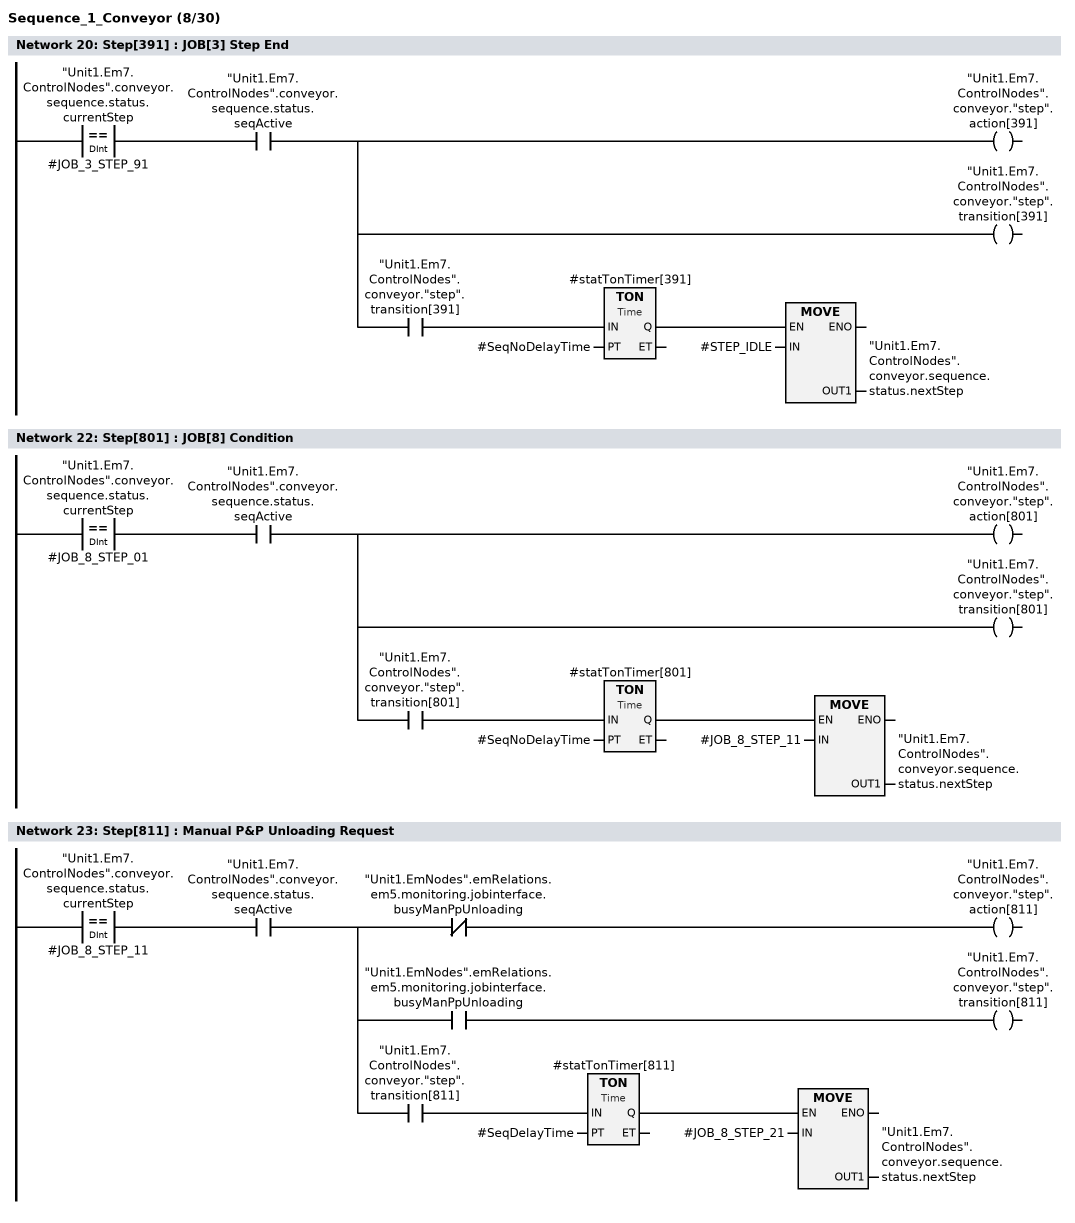
   RUNG wire#powerrail
      { S7_Templates := "SrcType := DInt" } EQ_Contact(in1 := "Unit1.Em7.ControlNodes".conveyor.sequence.status.currentStep, in2 := #JOB_3_STEP_91)
      Contact( "Unit1.Em7.ControlNodes".conveyor.sequence.status.seqActive )
      wire#w1
      Coil( "Unit1.Em7.ControlNodes".conveyor."step".action[391] )
   END_RUNG
   RUNG wire#w1
      Coil( "Unit1.Em7.ControlNodes".conveyor."step".transition[391] )
   END_RUNG
   RUNG wire#w1
      Contact( "Unit1.Em7.ControlNodes".conveyor."step".transition[391] )
      { S7_Templates := "time_type := Time" } #statTonTimer[391].TON(pt := #SeqNoDelayTime, et =>)
      Move(in := #STEP_IDLE, out1 => "Unit1.Em7.ControlNodes".conveyor.sequence.status.nextStep)
   END_RUNG
   // the same network as SCL:
   "Unit1.Em7.ControlNodes".conveyor."step".action[391] := ("Unit1.Em7.ControlNodes".conveyor.sequence.status.currentStep = #JOB_3_STEP_91) AND "Unit1.Em7.ControlNodes".conveyor.sequence.status.seqActive;
   "Unit1.Em7.ControlNodes".conveyor."step".transition[391] := ("Unit1.Em7.ControlNodes".conveyor.sequence.status.currentStep = #JOB_3_STEP_91) AND "Unit1.Em7.ControlNodes".conveyor.sequence.status.seqActive;
   #statTonTimer[391].TON(IN := ("Unit1.Em7.ControlNodes".conveyor.sequence.status.currentStep = #JOB_3_STEP_91) AND "Unit1.Em7.ControlNodes".conveyor.sequence.status.seqActive AND "Unit1.Em7.ControlNodes".conveyor."step".transition[391],
                          PT := #SeqNoDelayTime);
   IF #statTonTimer[391].Q THEN
       "Unit1.Em7.ControlNodes".conveyor.sequence.status.nextStep := #STEP_IDLE;
   END_IF;
END_REGION

REGION Network 21: ******************** JOB[8] REWORK REQ AUTO ********************
END_REGION

REGION Network 22: Step[801] : JOB[8] Condition
   RUNG wire#powerrail
      { S7_Templates := "SrcType := DInt" } EQ_Contact(in1 := "Unit1.Em7.ControlNodes".conveyor.sequence.status.currentStep, in2 := #JOB_8_STEP_01)
      Contact( "Unit1.Em7.ControlNodes".conveyor.sequence.status.seqActive )
      wire#w1
      Coil( "Unit1.Em7.ControlNodes".conveyor."step".action[801] )
   END_RUNG
   RUNG wire#w1
      Coil( "Unit1.Em7.ControlNodes".conveyor."step".transition[801] )
   END_RUNG
   RUNG wire#w1
      Contact( "Unit1.Em7.ControlNodes".conveyor."step".transition[801] )
      { S7_Templates := "time_type := Time" } #statTonTimer[801].TON(pt := #SeqNoDelayTime, et =>)
      Move(in := #JOB_8_STEP_11, out1 => "Unit1.Em7.ControlNodes".conveyor.sequence.status.nextStep)
   END_RUNG
   // the same network as SCL:
   "Unit1.Em7.ControlNodes".conveyor."step".action[801] := ("Unit1.Em7.ControlNodes".conveyor.sequence.status.currentStep = #JOB_8_STEP_01) AND "Unit1.Em7.ControlNodes".conveyor.sequence.status.seqActive;
   "Unit1.Em7.ControlNodes".conveyor."step".transition[801] := ("Unit1.Em7.ControlNodes".conveyor.sequence.status.currentStep = #JOB_8_STEP_01) AND "Unit1.Em7.ControlNodes".conveyor.sequence.status.seqActive;
   #statTonTimer[801].TON(IN := ("Unit1.Em7.ControlNodes".conveyor.sequence.status.currentStep = #JOB_8_STEP_01) AND "Unit1.Em7.ControlNodes".conveyor.sequence.status.seqActive AND "Unit1.Em7.ControlNodes".conveyor."step".transition[801],
                          PT := #SeqNoDelayTime);
   IF #statTonTimer[801].Q THEN
       "Unit1.Em7.ControlNodes".conveyor.sequence.status.nextStep := #JOB_8_STEP_11;
   END_IF;
END_REGION

REGION Network 23: Step[811] : Manual P&P Unloading Request
   RUNG wire#powerrail
      { S7_Templates := "SrcType := DInt" } EQ_Contact(in1 := "Unit1.Em7.ControlNodes".conveyor.sequence.status.currentStep, in2 := #JOB_8_STEP_11)
      Contact( "Unit1.Em7.ControlNodes".conveyor.sequence.status.seqActive )
      wire#w1
      I_Contact( "Unit1.EmNodes".emRelations.em5.monitoring.jobinterface.busyManPpUnloading )
      Coil( "Unit1.Em7.ControlNodes".conveyor."step".action[811] )
   END_RUNG
   RUNG wire#w1
      Contact( "Unit1.EmNodes".emRelations.em5.monitoring.jobinterface.busyManPpUnloading )
      Coil( "Unit1.Em7.ControlNodes".conveyor."step".transition[811] )
   END_RUNG
   RUNG wire#w1
      Contact( "Unit1.Em7.ControlNodes".conveyor."step".transition[811] )
      { S7_Templates := "time_type := Time" } #statTonTimer[811].TON(pt := #SeqDelayTime, et =>)
      Move(in := #JOB_8_STEP_21, out1 => "Unit1.Em7.ControlNodes".conveyor.sequence.status.nextStep)
   END_RUNG
   // the same network as SCL:
   #_w1 := ("Unit1.Em7.ControlNodes".conveyor.sequence.status.currentStep = #JOB_8_STEP_11) AND "Unit1.Em7.ControlNodes".conveyor.sequence.status.seqActive;
   "Unit1.Em7.ControlNodes".conveyor."step".action[811] := #_w1 AND NOT "Unit1.EmNodes".emRelations.em5.monitoring.jobinterface.busyManPpUnloading;
   "Unit1.Em7.ControlNodes".conveyor."step".transition[811] := #_w1 AND "Unit1.EmNodes".emRelations.em5.monitoring.jobinterface.busyManPpUnloading;
   #statTonTimer[811].TON(IN := #_w1 AND "Unit1.Em7.ControlNodes".conveyor."step".transition[811],
                          PT := #SeqDelayTime);
   IF #statTonTimer[811].Q THEN
       "Unit1.Em7.ControlNodes".conveyor.sequence.status.nextStep := #JOB_8_STEP_21;
   END_IF;
END_REGION

REGION Network 24: Step[821] : Manual P&P Unloading Done
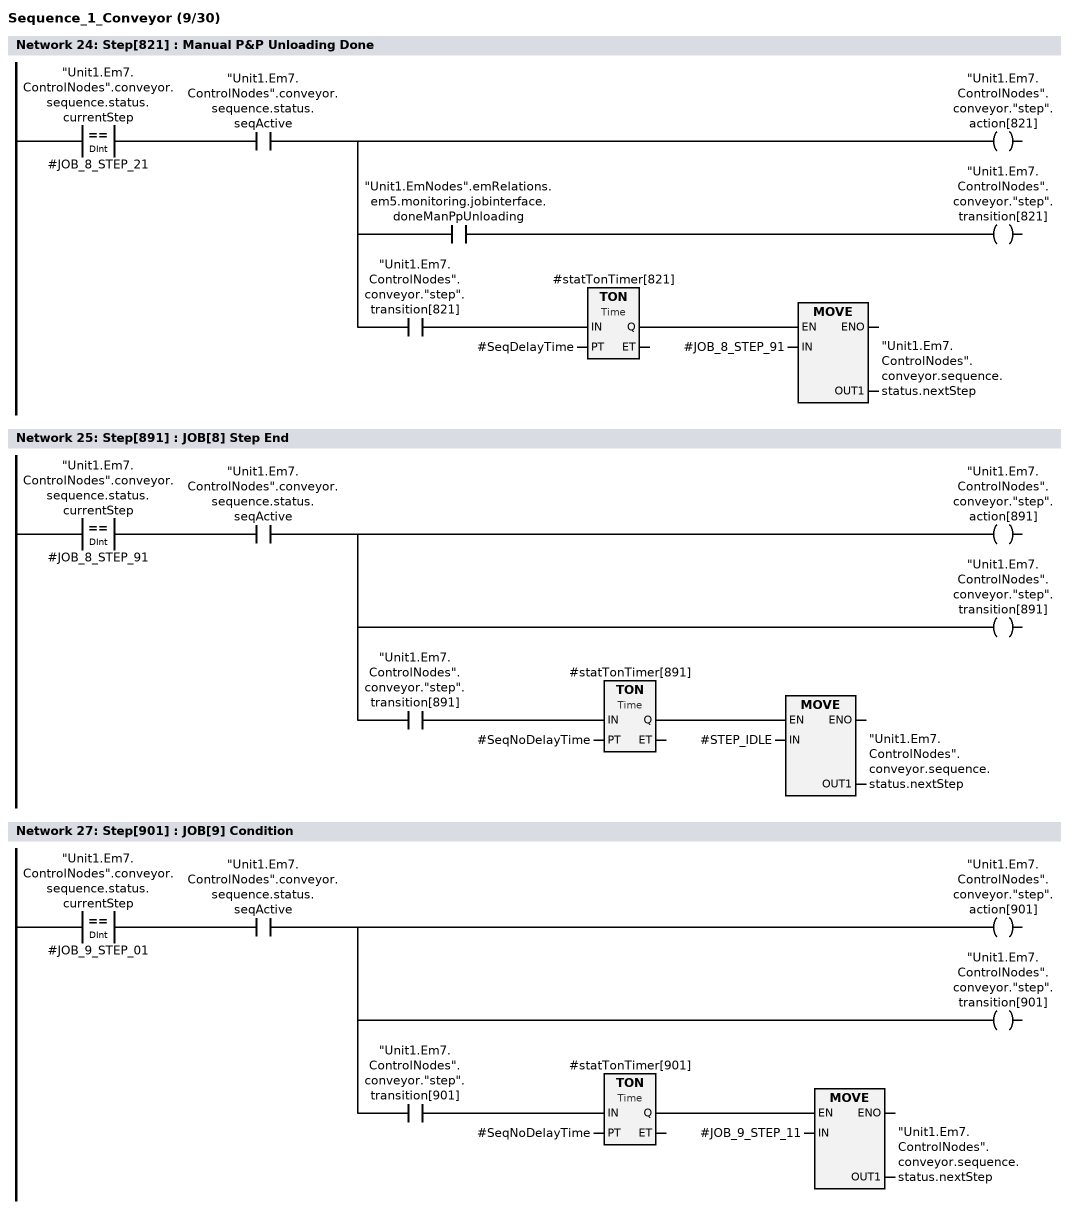
   RUNG wire#powerrail
      { S7_Templates := "SrcType := DInt" } EQ_Contact(in1 := "Unit1.Em7.ControlNodes".conveyor.sequence.status.currentStep, in2 := #JOB_8_STEP_21)
      Contact( "Unit1.Em7.ControlNodes".conveyor.sequence.status.seqActive )
      wire#w1
      Coil( "Unit1.Em7.ControlNodes".conveyor."step".action[821] )
   END_RUNG
   RUNG wire#w1
      Contact( "Unit1.EmNodes".emRelations.em5.monitoring.jobinterface.doneManPpUnloading )
      Coil( "Unit1.Em7.ControlNodes".conveyor."step".transition[821] )
   END_RUNG
   RUNG wire#w1
      Contact( "Unit1.Em7.ControlNodes".conveyor."step".transition[821] )
      { S7_Templates := "time_type := Time" } #statTonTimer[821].TON(pt := #SeqDelayTime, et =>)
      Move(in := #JOB_8_STEP_91, out1 => "Unit1.Em7.ControlNodes".conveyor.sequence.status.nextStep)
   END_RUNG
   // the same network as SCL:
   "Unit1.Em7.ControlNodes".conveyor."step".action[821] := ("Unit1.Em7.ControlNodes".conveyor.sequence.status.currentStep = #JOB_8_STEP_21) AND "Unit1.Em7.ControlNodes".conveyor.sequence.status.seqActive;
   "Unit1.Em7.ControlNodes".conveyor."step".transition[821] := ("Unit1.Em7.ControlNodes".conveyor.sequence.status.currentStep = #JOB_8_STEP_21) AND "Unit1.Em7.ControlNodes".conveyor.sequence.status.seqActive AND "Unit1.EmNodes".emRelations.em5.monitoring.jobinterface.doneManPpUnloading;
   #statTonTimer[821].TON(IN := ("Unit1.Em7.ControlNodes".conveyor.sequence.status.currentStep = #JOB_8_STEP_21) AND "Unit1.Em7.ControlNodes".conveyor.sequence.status.seqActive AND "Unit1.Em7.ControlNodes".conveyor."step".transition[821],
                          PT := #SeqDelayTime);
   IF #statTonTimer[821].Q THEN
       "Unit1.Em7.ControlNodes".conveyor.sequence.status.nextStep := #JOB_8_STEP_91;
   END_IF;
END_REGION

REGION Network 25: Step[891] : JOB[8] Step End
   RUNG wire#powerrail
      { S7_Templates := "SrcType := DInt" } EQ_Contact(in1 := "Unit1.Em7.ControlNodes".conveyor.sequence.status.currentStep, in2 := #JOB_8_STEP_91)
      Contact( "Unit1.Em7.ControlNodes".conveyor.sequence.status.seqActive )
      wire#w1
      Coil( "Unit1.Em7.ControlNodes".conveyor."step".action[891] )
   END_RUNG
   RUNG wire#w1
      Coil( "Unit1.Em7.ControlNodes".conveyor."step".transition[891] )
   END_RUNG
   RUNG wire#w1
      Contact( "Unit1.Em7.ControlNodes".conveyor."step".transition[891] )
      { S7_Templates := "time_type := Time" } #statTonTimer[891].TON(pt := #SeqNoDelayTime, et =>)
      Move(in := #STEP_IDLE, out1 => "Unit1.Em7.ControlNodes".conveyor.sequence.status.nextStep)
   END_RUNG
   // the same network as SCL:
   "Unit1.Em7.ControlNodes".conveyor."step".action[891] := ("Unit1.Em7.ControlNodes".conveyor.sequence.status.currentStep = #JOB_8_STEP_91) AND "Unit1.Em7.ControlNodes".conveyor.sequence.status.seqActive;
   "Unit1.Em7.ControlNodes".conveyor."step".transition[891] := ("Unit1.Em7.ControlNodes".conveyor.sequence.status.currentStep = #JOB_8_STEP_91) AND "Unit1.Em7.ControlNodes".conveyor.sequence.status.seqActive;
   #statTonTimer[891].TON(IN := ("Unit1.Em7.ControlNodes".conveyor.sequence.status.currentStep = #JOB_8_STEP_91) AND "Unit1.Em7.ControlNodes".conveyor.sequence.status.seqActive AND "Unit1.Em7.ControlNodes".conveyor."step".transition[891],
                          PT := #SeqNoDelayTime);
   IF #statTonTimer[891].Q THEN
       "Unit1.Em7.ControlNodes".conveyor.sequence.status.nextStep := #STEP_IDLE;
   END_IF;
END_REGION

REGION Network 26: ******************** JOB[9] VISION REQ AUTO ********************
END_REGION

REGION Network 27: Step[901] : JOB[9] Condition
   RUNG wire#powerrail
      { S7_Templates := "SrcType := DInt" } EQ_Contact(in1 := "Unit1.Em7.ControlNodes".conveyor.sequence.status.currentStep, in2 := #JOB_9_STEP_01)
      Contact( "Unit1.Em7.ControlNodes".conveyor.sequence.status.seqActive )
      wire#w1
      Coil( "Unit1.Em7.ControlNodes".conveyor."step".action[901] )
   END_RUNG
   RUNG wire#w1
      Coil( "Unit1.Em7.ControlNodes".conveyor."step".transition[901] )
   END_RUNG
   RUNG wire#w1
      Contact( "Unit1.Em7.ControlNodes".conveyor."step".transition[901] )
      { S7_Templates := "time_type := Time" } #statTonTimer[901].TON(pt := #SeqNoDelayTime, et =>)
      Move(in := #JOB_9_STEP_11, out1 => "Unit1.Em7.ControlNodes".conveyor.sequence.status.nextStep)
   END_RUNG
   // the same network as SCL:
   "Unit1.Em7.ControlNodes".conveyor."step".action[901] := ("Unit1.Em7.ControlNodes".conveyor.sequence.status.currentStep = #JOB_9_STEP_01) AND "Unit1.Em7.ControlNodes".conveyor.sequence.status.seqActive;
   "Unit1.Em7.ControlNodes".conveyor."step".transition[901] := ("Unit1.Em7.ControlNodes".conveyor.sequence.status.currentStep = #JOB_9_STEP_01) AND "Unit1.Em7.ControlNodes".conveyor.sequence.status.seqActive;
   #statTonTimer[901].TON(IN := ("Unit1.Em7.ControlNodes".conveyor.sequence.status.currentStep = #JOB_9_STEP_01) AND "Unit1.Em7.ControlNodes".conveyor.sequence.status.seqActive AND "Unit1.Em7.ControlNodes".conveyor."step".transition[901],
                          PT := #SeqNoDelayTime);
   IF #statTonTimer[901].Q THEN
       "Unit1.Em7.ControlNodes".conveyor.sequence.status.nextStep := #JOB_9_STEP_11;
   END_IF;
END_REGION

REGION Network 28: Step[911] : Vision Inspection Request
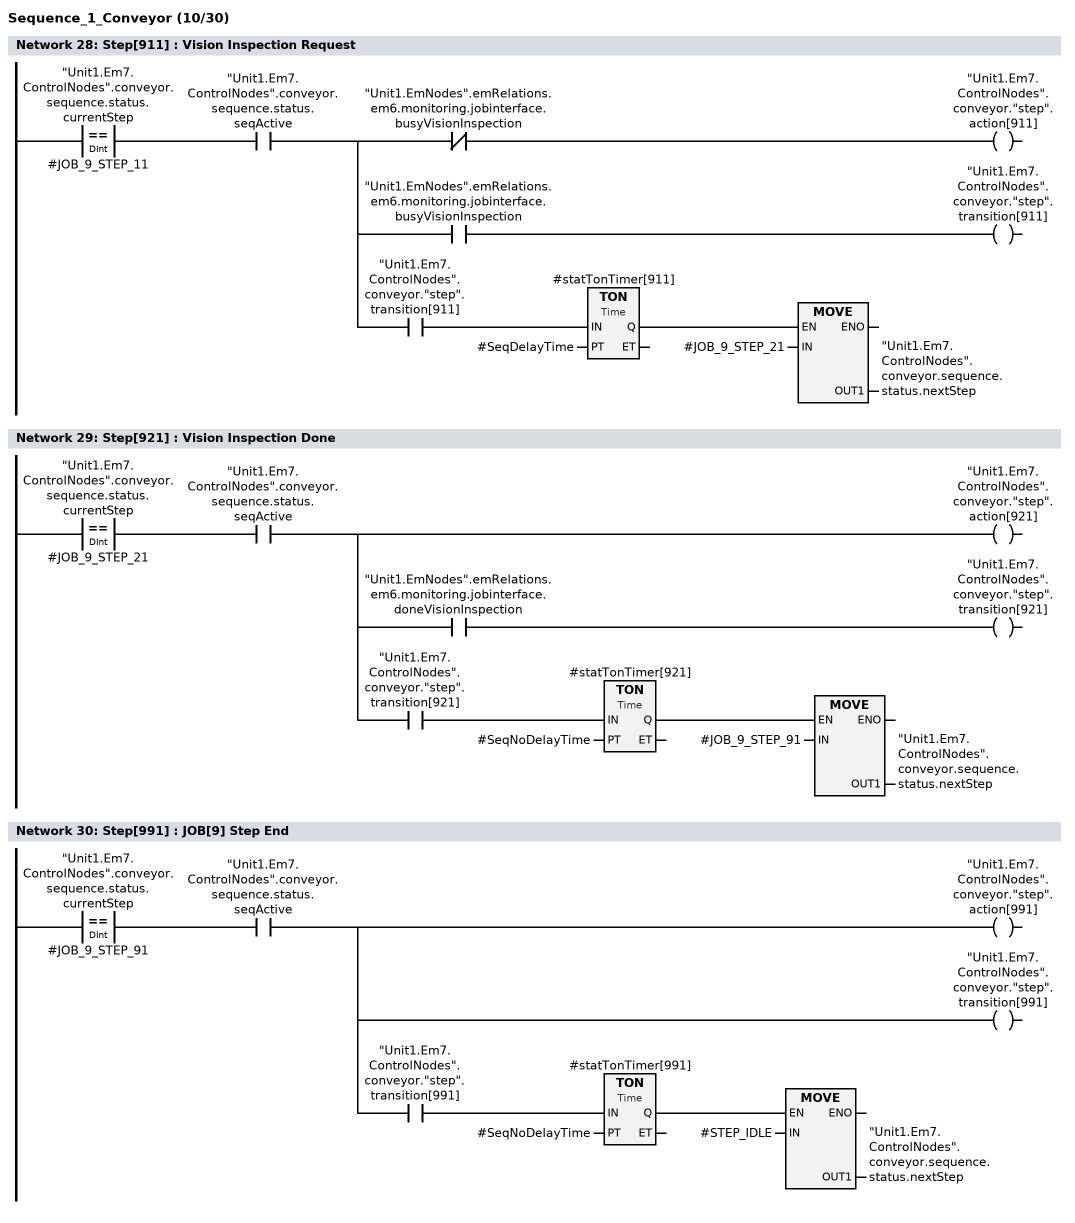
   RUNG wire#powerrail
      { S7_Templates := "SrcType := DInt" } EQ_Contact(in1 := "Unit1.Em7.ControlNodes".conveyor.sequence.status.currentStep, in2 := #JOB_9_STEP_11)
      Contact( "Unit1.Em7.ControlNodes".conveyor.sequence.status.seqActive )
      wire#w1
      I_Contact( "Unit1.EmNodes".emRelations.em6.monitoring.jobinterface.busyVisionInspection )
      Coil( "Unit1.Em7.ControlNodes".conveyor."step".action[911] )
   END_RUNG
   RUNG wire#w1
      Contact( "Unit1.EmNodes".emRelations.em6.monitoring.jobinterface.busyVisionInspection )
      Coil( "Unit1.Em7.ControlNodes".conveyor."step".transition[911] )
   END_RUNG
   RUNG wire#w1
      Contact( "Unit1.Em7.ControlNodes".conveyor."step".transition[911] )
      { S7_Templates := "time_type := Time" } #statTonTimer[911].TON(pt := #SeqDelayTime, et =>)
      Move(in := #JOB_9_STEP_21, out1 => "Unit1.Em7.ControlNodes".conveyor.sequence.status.nextStep)
   END_RUNG
   // the same network as SCL:
   #_w1 := ("Unit1.Em7.ControlNodes".conveyor.sequence.status.currentStep = #JOB_9_STEP_11) AND "Unit1.Em7.ControlNodes".conveyor.sequence.status.seqActive;
   "Unit1.Em7.ControlNodes".conveyor."step".action[911] := #_w1 AND NOT "Unit1.EmNodes".emRelations.em6.monitoring.jobinterface.busyVisionInspection;
   "Unit1.Em7.ControlNodes".conveyor."step".transition[911] := #_w1 AND "Unit1.EmNodes".emRelations.em6.monitoring.jobinterface.busyVisionInspection;
   #statTonTimer[911].TON(IN := #_w1 AND "Unit1.Em7.ControlNodes".conveyor."step".transition[911],
                          PT := #SeqDelayTime);
   IF #statTonTimer[911].Q THEN
       "Unit1.Em7.ControlNodes".conveyor.sequence.status.nextStep := #JOB_9_STEP_21;
   END_IF;
END_REGION

REGION Network 29: Step[921] : Vision Inspection Done
   RUNG wire#powerrail
      { S7_Templates := "SrcType := DInt" } EQ_Contact(in1 := "Unit1.Em7.ControlNodes".conveyor.sequence.status.currentStep, in2 := #JOB_9_STEP_21)
      Contact( "Unit1.Em7.ControlNodes".conveyor.sequence.status.seqActive )
      wire#w1
      Coil( "Unit1.Em7.ControlNodes".conveyor."step".action[921] )
   END_RUNG
   RUNG wire#w1
      Contact( "Unit1.EmNodes".emRelations.em6.monitoring.jobinterface.doneVisionInspection )
      Coil( "Unit1.Em7.ControlNodes".conveyor."step".transition[921] )
   END_RUNG
   RUNG wire#w1
      Contact( "Unit1.Em7.ControlNodes".conveyor."step".transition[921] )
      { S7_Templates := "time_type := Time" } #statTonTimer[921].TON(pt := #SeqNoDelayTime, et =>)
      Move(in := #JOB_9_STEP_91, out1 => "Unit1.Em7.ControlNodes".conveyor.sequence.status.nextStep)
   END_RUNG
   // the same network as SCL:
   "Unit1.Em7.ControlNodes".conveyor."step".action[921] := ("Unit1.Em7.ControlNodes".conveyor.sequence.status.currentStep = #JOB_9_STEP_21) AND "Unit1.Em7.ControlNodes".conveyor.sequence.status.seqActive;
   "Unit1.Em7.ControlNodes".conveyor."step".transition[921] := ("Unit1.Em7.ControlNodes".conveyor.sequence.status.currentStep = #JOB_9_STEP_21) AND "Unit1.Em7.ControlNodes".conveyor.sequence.status.seqActive AND "Unit1.EmNodes".emRelations.em6.monitoring.jobinterface.doneVisionInspection;
   #statTonTimer[921].TON(IN := ("Unit1.Em7.ControlNodes".conveyor.sequence.status.currentStep = #JOB_9_STEP_21) AND "Unit1.Em7.ControlNodes".conveyor.sequence.status.seqActive AND "Unit1.Em7.ControlNodes".conveyor."step".transition[921],
                          PT := #SeqNoDelayTime);
   IF #statTonTimer[921].Q THEN
       "Unit1.Em7.ControlNodes".conveyor.sequence.status.nextStep := #JOB_9_STEP_91;
   END_IF;
END_REGION

REGION Network 30: Step[991] : JOB[9] Step End
   RUNG wire#powerrail
      { S7_Templates := "SrcType := DInt" } EQ_Contact(in1 := "Unit1.Em7.ControlNodes".conveyor.sequence.status.currentStep, in2 := #JOB_9_STEP_91)
      Contact( "Unit1.Em7.ControlNodes".conveyor.sequence.status.seqActive )
      wire#w1
      Coil( "Unit1.Em7.ControlNodes".conveyor."step".action[991] )
   END_RUNG
   RUNG wire#w1
      Coil( "Unit1.Em7.ControlNodes".conveyor."step".transition[991] )
   END_RUNG
   RUNG wire#w1
      Contact( "Unit1.Em7.ControlNodes".conveyor."step".transition[991] )
      { S7_Templates := "time_type := Time" } #statTonTimer[991].TON(pt := #SeqNoDelayTime, et =>)
      Move(in := #STEP_IDLE, out1 => "Unit1.Em7.ControlNodes".conveyor.sequence.status.nextStep)
   END_RUNG
   // the same network as SCL:
   "Unit1.Em7.ControlNodes".conveyor."step".action[991] := ("Unit1.Em7.ControlNodes".conveyor.sequence.status.currentStep = #JOB_9_STEP_91) AND "Unit1.Em7.ControlNodes".conveyor.sequence.status.seqActive;
   "Unit1.Em7.ControlNodes".conveyor."step".transition[991] := ("Unit1.Em7.ControlNodes".conveyor.sequence.status.currentStep = #JOB_9_STEP_91) AND "Unit1.Em7.ControlNodes".conveyor.sequence.status.seqActive;
   #statTonTimer[991].TON(IN := ("Unit1.Em7.ControlNodes".conveyor.sequence.status.currentStep = #JOB_9_STEP_91) AND "Unit1.Em7.ControlNodes".conveyor.sequence.status.seqActive AND "Unit1.Em7.ControlNodes".conveyor."step".transition[991],
                          PT := #SeqNoDelayTime);
   IF #statTonTimer[991].Q THEN
       "Unit1.Em7.ControlNodes".conveyor.sequence.status.nextStep := #STEP_IDLE;
   END_IF;
END_REGION

REGION Network 31: ******************** JOB[10] ReelCut GAUGE R&R AUTO ********************
END_REGION

REGION Network 32: Step[1001] : JOB[10] Condition
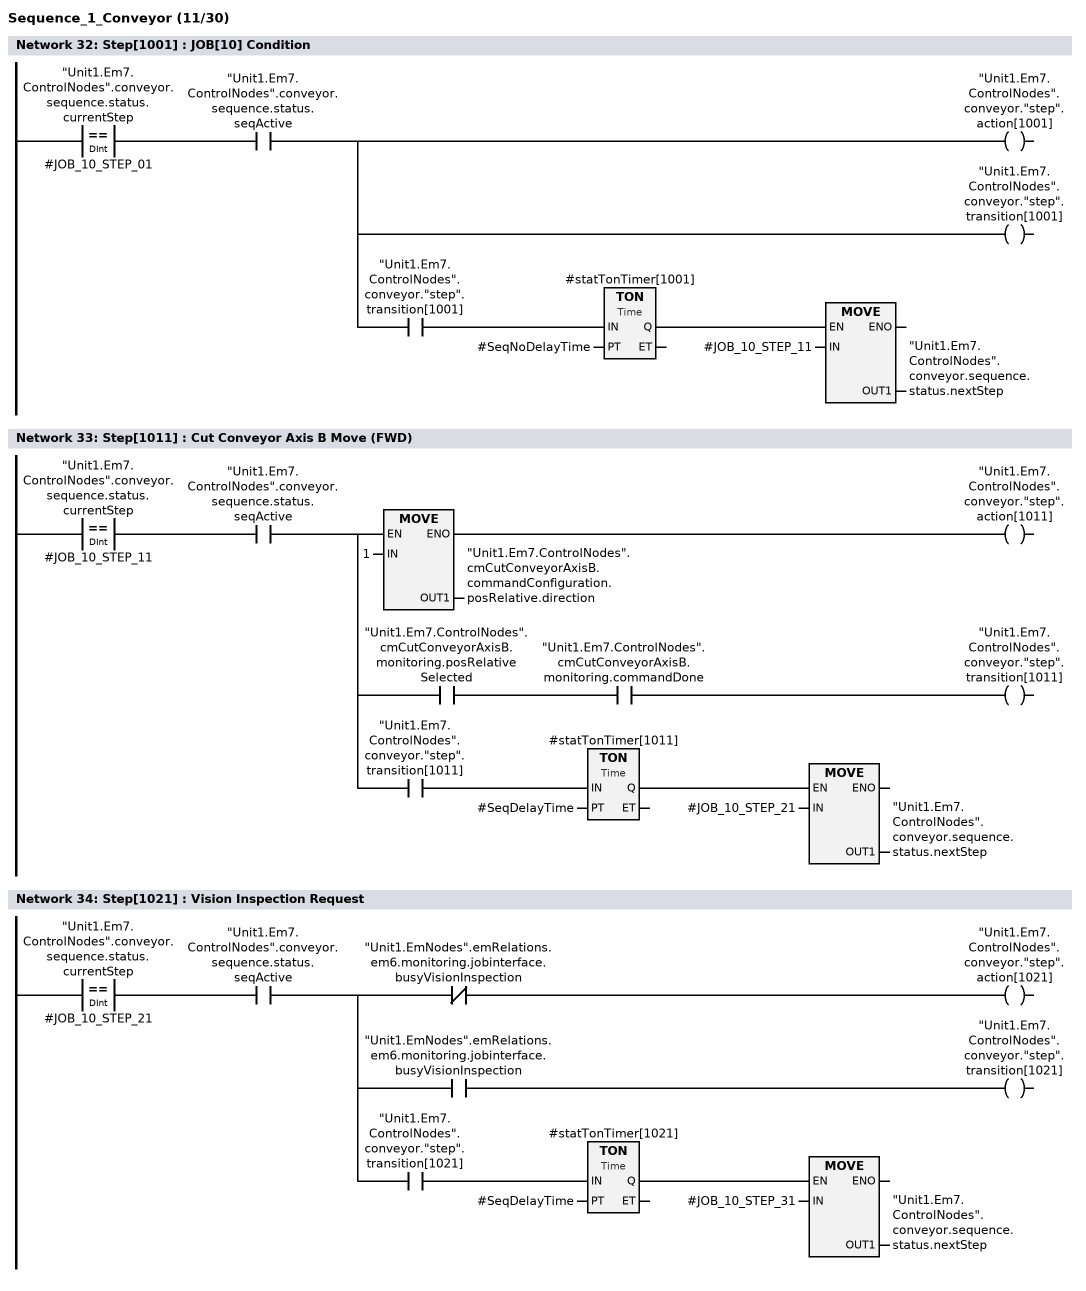
   RUNG wire#powerrail
      { S7_Templates := "SrcType := DInt" } EQ_Contact(in1 := "Unit1.Em7.ControlNodes".conveyor.sequence.status.currentStep, in2 := #JOB_10_STEP_01)
      Contact( "Unit1.Em7.ControlNodes".conveyor.sequence.status.seqActive )
      wire#w1
      Coil( "Unit1.Em7.ControlNodes".conveyor."step".action[1001] )
   END_RUNG
   RUNG wire#w1
      Coil( "Unit1.Em7.ControlNodes".conveyor."step".transition[1001] )
   END_RUNG
   RUNG wire#w1
      Contact( "Unit1.Em7.ControlNodes".conveyor."step".transition[1001] )
      { S7_Templates := "time_type := Time" } #statTonTimer[1001].TON(pt := #SeqNoDelayTime, et =>)
      Move(in := #JOB_10_STEP_11, out1 => "Unit1.Em7.ControlNodes".conveyor.sequence.status.nextStep)
   END_RUNG
   // the same network as SCL:
   "Unit1.Em7.ControlNodes".conveyor."step".action[1001] := ("Unit1.Em7.ControlNodes".conveyor.sequence.status.currentStep = #JOB_10_STEP_01) AND "Unit1.Em7.ControlNodes".conveyor.sequence.status.seqActive;
   "Unit1.Em7.ControlNodes".conveyor."step".transition[1001] := ("Unit1.Em7.ControlNodes".conveyor.sequence.status.currentStep = #JOB_10_STEP_01) AND "Unit1.Em7.ControlNodes".conveyor.sequence.status.seqActive;
   #statTonTimer[1001].TON(IN := ("Unit1.Em7.ControlNodes".conveyor.sequence.status.currentStep = #JOB_10_STEP_01) AND "Unit1.Em7.ControlNodes".conveyor.sequence.status.seqActive AND "Unit1.Em7.ControlNodes".conveyor."step".transition[1001],
                           PT := #SeqNoDelayTime);
   IF #statTonTimer[1001].Q THEN
       "Unit1.Em7.ControlNodes".conveyor.sequence.status.nextStep := #JOB_10_STEP_11;
   END_IF;
END_REGION

REGION Network 33: Step[1011] : Cut Conveyor Axis B Move (FWD)
   RUNG wire#powerrail
      { S7_Templates := "SrcType := DInt" } EQ_Contact(in1 := "Unit1.Em7.ControlNodes".conveyor.sequence.status.currentStep, in2 := #JOB_10_STEP_11)
      Contact( "Unit1.Em7.ControlNodes".conveyor.sequence.status.seqActive )
      wire#w1
      Move(in := 1, out1 => "Unit1.Em7.ControlNodes".cmCutConveyorAxisB.commandConfiguration.posRelative.direction)
      Coil( "Unit1.Em7.ControlNodes".conveyor."step".action[1011] )
   END_RUNG
   RUNG wire#w1
      Contact( "Unit1.Em7.ControlNodes".cmCutConveyorAxisB.monitoring.posRelativeSelected )
      Contact( "Unit1.Em7.ControlNodes".cmCutConveyorAxisB.monitoring.commandDone )
      Coil( "Unit1.Em7.ControlNodes".conveyor."step".transition[1011] )
   END_RUNG
   RUNG wire#w1
      Contact( "Unit1.Em7.ControlNodes".conveyor."step".transition[1011] )
      { S7_Templates := "time_type := Time" } #statTonTimer[1011].TON(pt := #SeqDelayTime, et =>)
      Move(in := #JOB_10_STEP_21, out1 => "Unit1.Em7.ControlNodes".conveyor.sequence.status.nextStep)
   END_RUNG
   // the same network as SCL:
   #_w1 := ("Unit1.Em7.ControlNodes".conveyor.sequence.status.currentStep = #JOB_10_STEP_11) AND "Unit1.Em7.ControlNodes".conveyor.sequence.status.seqActive;
   IF #_w1 THEN
       "Unit1.Em7.ControlNodes".cmCutConveyorAxisB.commandConfiguration.posRelative.direction := 1;
   END_IF;
   "Unit1.Em7.ControlNodes".conveyor."step".action[1011] := #_w1;
   "Unit1.Em7.ControlNodes".conveyor."step".transition[1011] := #_w1 AND "Unit1.Em7.ControlNodes".cmCutConveyorAxisB.monitoring.posRelativeSelected AND "Unit1.Em7.ControlNodes".cmCutConveyorAxisB.monitoring.commandDone;
   #statTonTimer[1011].TON(IN := #_w1 AND "Unit1.Em7.ControlNodes".conveyor."step".transition[1011],
                           PT := #SeqDelayTime);
   IF #statTonTimer[1011].Q THEN
       "Unit1.Em7.ControlNodes".conveyor.sequence.status.nextStep := #JOB_10_STEP_21;
   END_IF;
END_REGION

REGION Network 34: Step[1021] : Vision Inspection Request
   RUNG wire#powerrail
      { S7_Templates := "SrcType := DInt" } EQ_Contact(in1 := "Unit1.Em7.ControlNodes".conveyor.sequence.status.currentStep, in2 := #JOB_10_STEP_21)
      Contact( "Unit1.Em7.ControlNodes".conveyor.sequence.status.seqActive )
      wire#w1
      I_Contact( "Unit1.EmNodes".emRelations.em6.monitoring.jobinterface.busyVisionInspection )
      Coil( "Unit1.Em7.ControlNodes".conveyor."step".action[1021] )
   END_RUNG
   RUNG wire#w1
      Contact( "Unit1.EmNodes".emRelations.em6.monitoring.jobinterface.busyVisionInspection )
      Coil( "Unit1.Em7.ControlNodes".conveyor."step".transition[1021] )
   END_RUNG
   RUNG wire#w1
      Contact( "Unit1.Em7.ControlNodes".conveyor."step".transition[1021] )
      { S7_Templates := "time_type := Time" } #statTonTimer[1021].TON(pt := #SeqDelayTime, et =>)
      Move(in := #JOB_10_STEP_31, out1 => "Unit1.Em7.ControlNodes".conveyor.sequence.status.nextStep)
   END_RUNG
   // the same network as SCL:
   #_w1 := ("Unit1.Em7.ControlNodes".conveyor.sequence.status.currentStep = #JOB_10_STEP_21) AND "Unit1.Em7.ControlNodes".conveyor.sequence.status.seqActive;
   "Unit1.Em7.ControlNodes".conveyor."step".action[1021] := #_w1 AND NOT "Unit1.EmNodes".emRelations.em6.monitoring.jobinterface.busyVisionInspection;
   "Unit1.Em7.ControlNodes".conveyor."step".transition[1021] := #_w1 AND "Unit1.EmNodes".emRelations.em6.monitoring.jobinterface.busyVisionInspection;
   #statTonTimer[1021].TON(IN := #_w1 AND "Unit1.Em7.ControlNodes".conveyor."step".transition[1021],
                           PT := #SeqDelayTime);
   IF #statTonTimer[1021].Q THEN
       "Unit1.Em7.ControlNodes".conveyor.sequence.status.nextStep := #JOB_10_STEP_31;
   END_IF;
END_REGION

REGION Network 35: Step[1031] : Vision Inspection Done
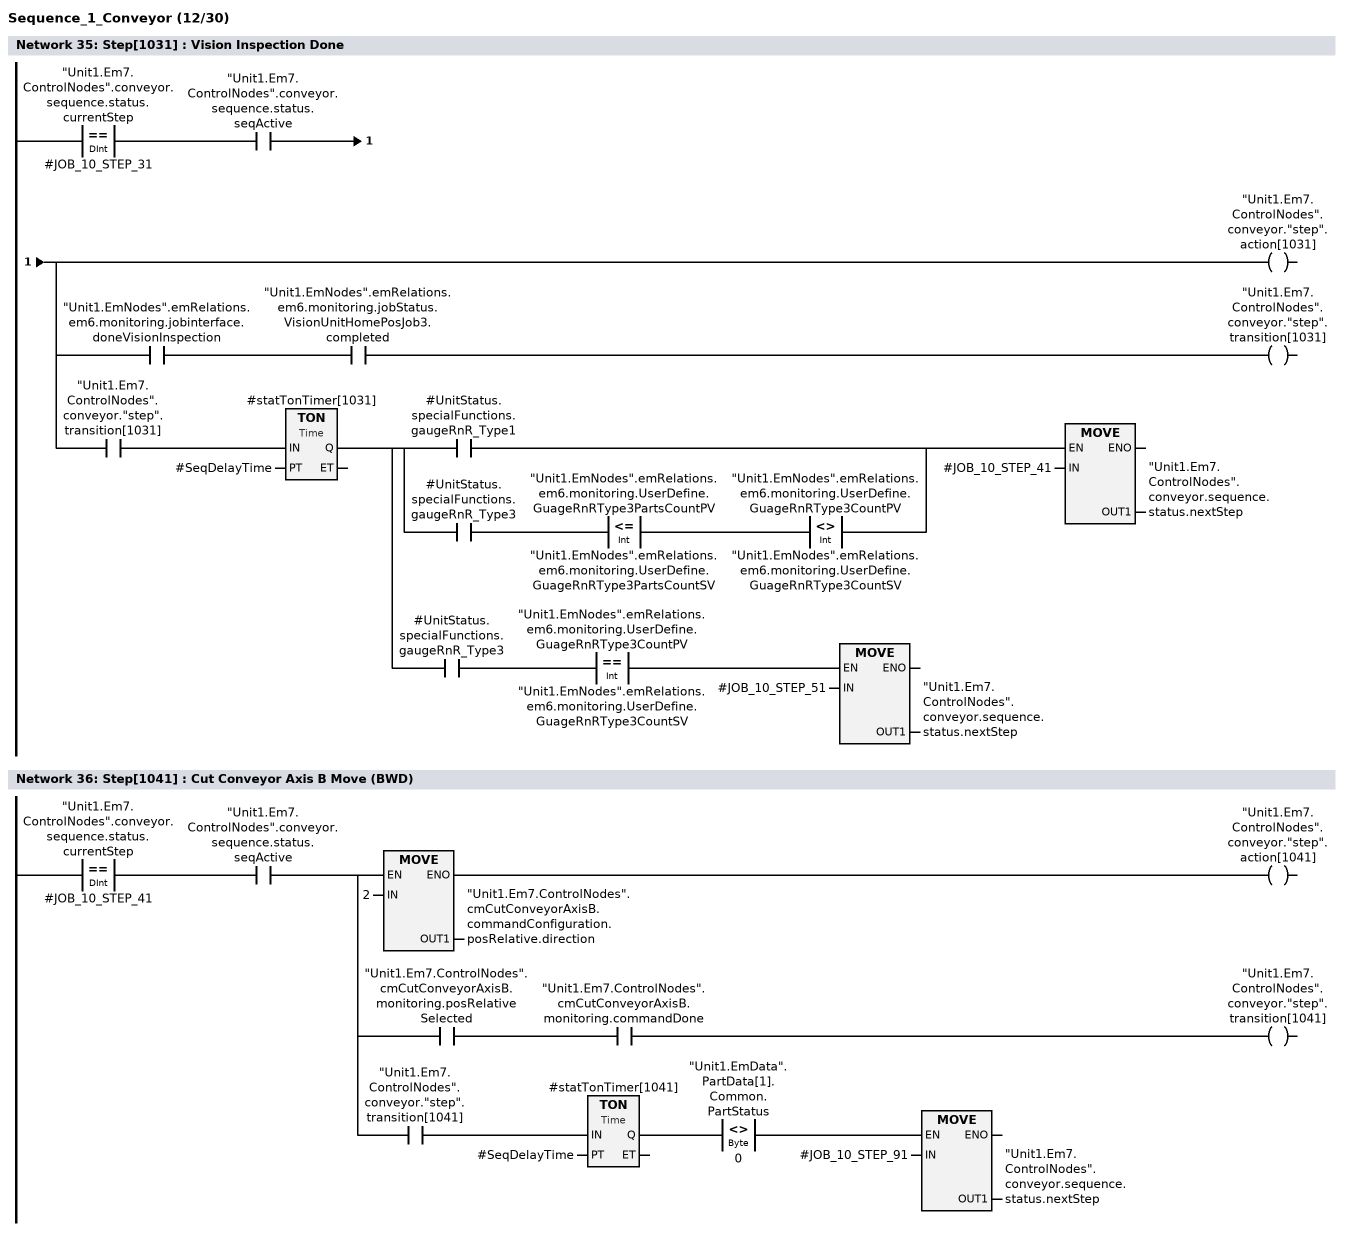
   RUNG wire#powerrail
      { S7_Templates := "SrcType := DInt" } EQ_Contact(in1 := "Unit1.Em7.ControlNodes".conveyor.sequence.status.currentStep, in2 := #JOB_10_STEP_31)
      Contact( "Unit1.Em7.ControlNodes".conveyor.sequence.status.seqActive )
      wire#w1
      Coil( "Unit1.Em7.ControlNodes".conveyor."step".action[1031] )
   END_RUNG
   RUNG wire#w1
      Contact( "Unit1.EmNodes".emRelations.em6.monitoring.jobinterface.doneVisionInspection )
      Contact( "Unit1.EmNodes".emRelations.em6.monitoring.jobStatus.VisionUnitHomePosJob3.completed )
      Coil( "Unit1.Em7.ControlNodes".conveyor."step".transition[1031] )
   END_RUNG
   RUNG wire#w1
      Contact( "Unit1.Em7.ControlNodes".conveyor."step".transition[1031] )
      { S7_Templates := "time_type := Time" } #statTonTimer[1031].TON(pt := #SeqDelayTime, et =>)
      wire#w2
      Contact( #UnitStatus.specialFunctions.gaugeRnR_Type1 )
      wire#w3
      Move(in := #JOB_10_STEP_41, out1 => "Unit1.Em7.ControlNodes".conveyor.sequence.status.nextStep)
   END_RUNG
   RUNG wire#w2
      Contact( #UnitStatus.specialFunctions.gaugeRnR_Type3 )
      { S7_Templates := "SrcType := Int" } LE_Contact(in1 := "Unit1.EmNodes".emRelations.em6.monitoring.UserDefine.GuageRnRType3PartsCountPV, in2 := "Unit1.EmNodes".emRelations.em6.monitoring.UserDefine.GuageRnRType3PartsCountSV)
      { S7_Templates := "SrcType := Int" } NE_Contact(in1 := "Unit1.EmNodes".emRelations.em6.monitoring.UserDefine.GuageRnRType3CountPV, in2 := "Unit1.EmNodes".emRelations.em6.monitoring.UserDefine.GuageRnRType3CountSV)
   END_RUNG wire#w3
   RUNG wire#w2
      Contact( #UnitStatus.specialFunctions.gaugeRnR_Type3 )
      { S7_Templates := "SrcType := Int" } EQ_Contact(in1 := "Unit1.EmNodes".emRelations.em6.monitoring.UserDefine.GuageRnRType3CountPV, in2 := "Unit1.EmNodes".emRelations.em6.monitoring.UserDefine.GuageRnRType3CountSV)
      Move(in := #JOB_10_STEP_51, out1 => "Unit1.Em7.ControlNodes".conveyor.sequence.status.nextStep)
   END_RUNG
   // the same network as SCL:
   "Unit1.Em7.ControlNodes".conveyor."step".action[1031] := ("Unit1.Em7.ControlNodes".conveyor.sequence.status.currentStep = #JOB_10_STEP_31) AND "Unit1.Em7.ControlNodes".conveyor.sequence.status.seqActive;
   "Unit1.Em7.ControlNodes".conveyor."step".transition[1031] := ("Unit1.Em7.ControlNodes".conveyor.sequence.status.currentStep = #JOB_10_STEP_31) AND "Unit1.Em7.ControlNodes".conveyor.sequence.status.seqActive AND "Unit1.EmNodes".emRelations.em6.monitoring.jobinterface.doneVisionInspection AND "Unit1.EmNodes".emRelations.em6.monitoring.jobStatus.VisionUnitHomePosJob3.completed;
   #statTonTimer[1031].TON(IN := ("Unit1.Em7.ControlNodes".conveyor.sequence.status.currentStep = #JOB_10_STEP_31) AND "Unit1.Em7.ControlNodes".conveyor.sequence.status.seqActive AND "Unit1.Em7.ControlNodes".conveyor."step".transition[1031],
                           PT := #SeqDelayTime);
   IF #statTonTimer[1031].Q AND (#UnitStatus.specialFunctions.gaugeRnR_Type1 OR (#UnitStatus.specialFunctions.gaugeRnR_Type3 AND ("Unit1.EmNodes".emRelations.em6.monitoring.UserDefine.GuageRnRType3PartsCountPV <= "Unit1.EmNodes".emRelations.em6.monitoring.UserDefine.GuageRnRType3PartsCountSV) AND ("Unit1.EmNodes".emRelations.em6.monitoring.UserDefine.GuageRnRType3CountPV <> "Unit1.EmNodes".emRelations.em6.monitoring.UserDefine.GuageRnRType3CountSV))) THEN
       "Unit1.Em7.ControlNodes".conveyor.sequence.status.nextStep := #JOB_10_STEP_41;
   END_IF;
   IF #statTonTimer[1031].Q AND #UnitStatus.specialFunctions.gaugeRnR_Type3 AND ("Unit1.EmNodes".emRelations.em6.monitoring.UserDefine.GuageRnRType3CountPV = "Unit1.EmNodes".emRelations.em6.monitoring.UserDefine.GuageRnRType3CountSV) THEN
       "Unit1.Em7.ControlNodes".conveyor.sequence.status.nextStep := #JOB_10_STEP_51;
   END_IF;
END_REGION

REGION Network 36: Step[1041] : Cut Conveyor Axis B Move (BWD)
   RUNG wire#powerrail
      { S7_Templates := "SrcType := DInt" } EQ_Contact(in1 := "Unit1.Em7.ControlNodes".conveyor.sequence.status.currentStep, in2 := #JOB_10_STEP_41)
      Contact( "Unit1.Em7.ControlNodes".conveyor.sequence.status.seqActive )
      wire#w1
      Move(in := 2, out1 => "Unit1.Em7.ControlNodes".cmCutConveyorAxisB.commandConfiguration.posRelative.direction)
      Coil( "Unit1.Em7.ControlNodes".conveyor."step".action[1041] )
   END_RUNG
   RUNG wire#w1
      Contact( "Unit1.Em7.ControlNodes".cmCutConveyorAxisB.monitoring.posRelativeSelected )
      Contact( "Unit1.Em7.ControlNodes".cmCutConveyorAxisB.monitoring.commandDone )
      Coil( "Unit1.Em7.ControlNodes".conveyor."step".transition[1041] )
   END_RUNG
   RUNG wire#w1
      Contact( "Unit1.Em7.ControlNodes".conveyor."step".transition[1041] )
      { S7_Templates := "time_type := Time" } #statTonTimer[1041].TON(pt := #SeqDelayTime, et =>)
      { S7_Templates := "SrcType := Byte" } NE_Contact(in1 := "Unit1.EmData".PartData[1].Common.PartStatus, in2 := 0)
      Move(in := #JOB_10_STEP_91, out1 => "Unit1.Em7.ControlNodes".conveyor.sequence.status.nextStep)
   END_RUNG
   // the same network as SCL:
   #_w1 := ("Unit1.Em7.ControlNodes".conveyor.sequence.status.currentStep = #JOB_10_STEP_41) AND "Unit1.Em7.ControlNodes".conveyor.sequence.status.seqActive;
   IF #_w1 THEN
       "Unit1.Em7.ControlNodes".cmCutConveyorAxisB.commandConfiguration.posRelative.direction := 2;
   END_IF;
   "Unit1.Em7.ControlNodes".conveyor."step".action[1041] := #_w1;
   "Unit1.Em7.ControlNodes".conveyor."step".transition[1041] := #_w1 AND "Unit1.Em7.ControlNodes".cmCutConveyorAxisB.monitoring.posRelativeSelected AND "Unit1.Em7.ControlNodes".cmCutConveyorAxisB.monitoring.commandDone;
   #statTonTimer[1041].TON(IN := #_w1 AND "Unit1.Em7.ControlNodes".conveyor."step".transition[1041],
                           PT := #SeqDelayTime);
   IF #statTonTimer[1041].Q AND ("Unit1.EmData".PartData[1].Common.PartStatus <> 0) THEN
       "Unit1.Em7.ControlNodes".conveyor.sequence.status.nextStep := #JOB_10_STEP_91;
   END_IF;
END_REGION

REGION Network 37: Step[1051] : Conveyor Empty Semi Auto
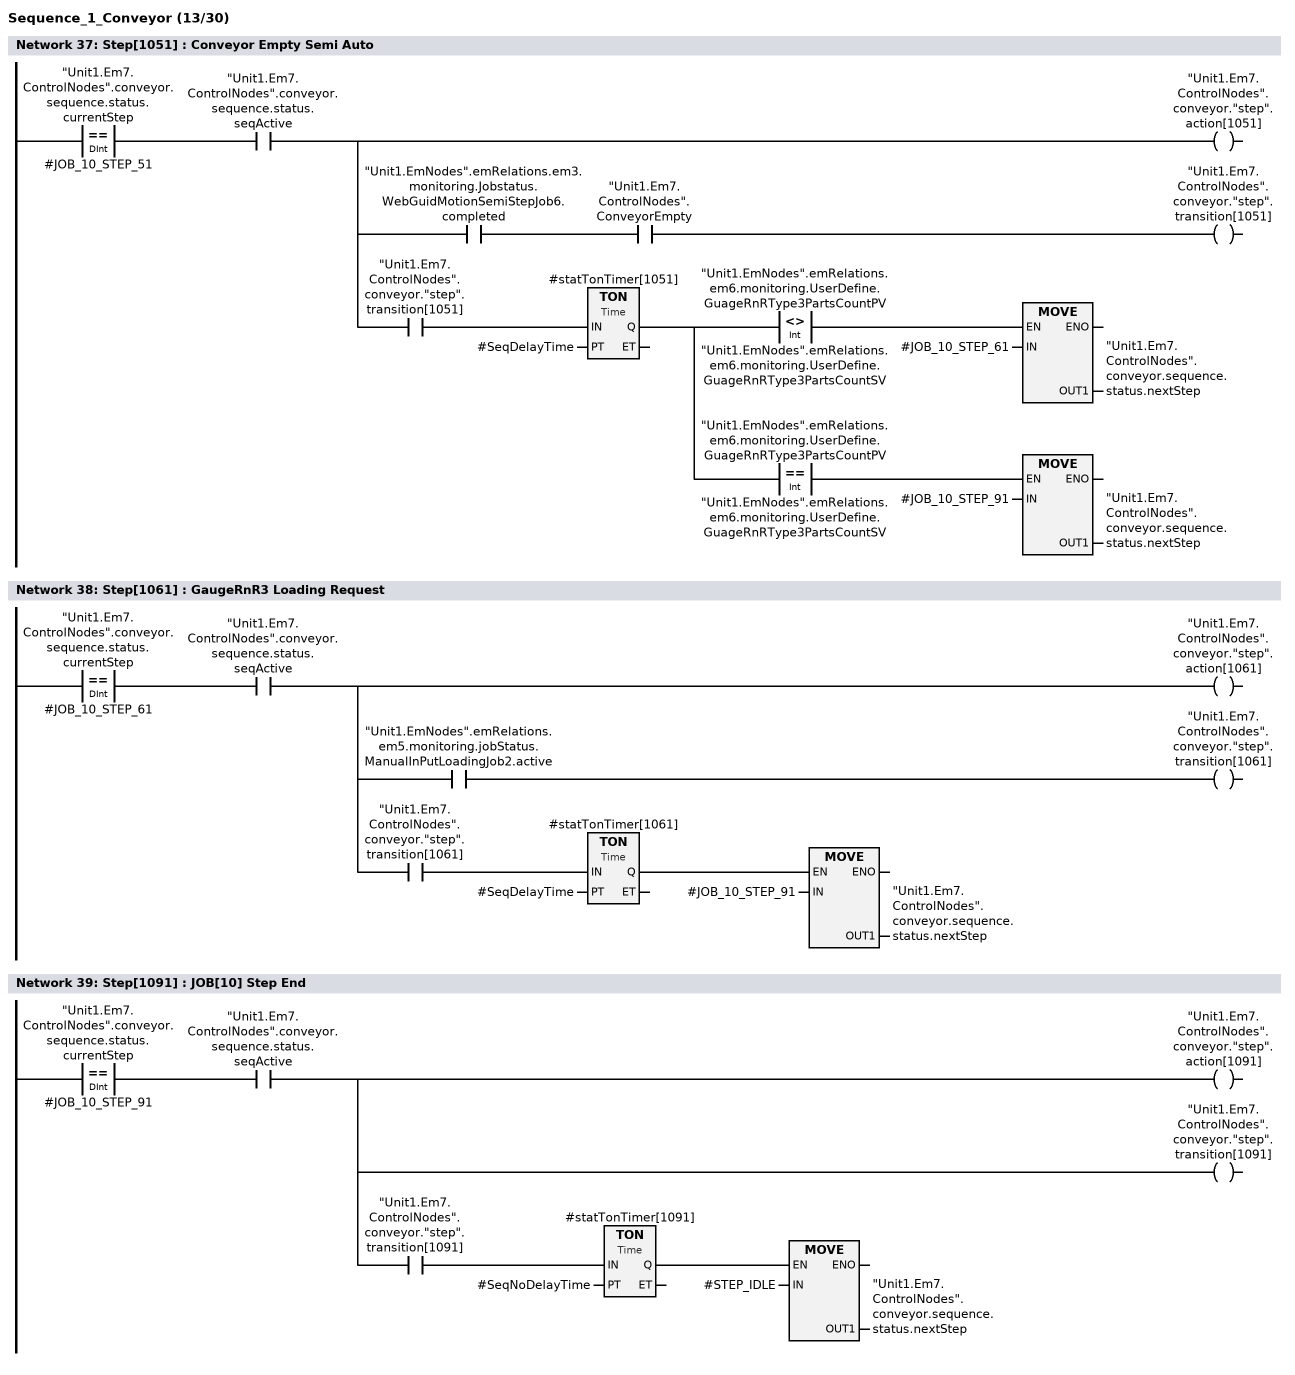
   RUNG wire#powerrail
      { S7_Templates := "SrcType := DInt" } EQ_Contact(in1 := "Unit1.Em7.ControlNodes".conveyor.sequence.status.currentStep, in2 := #JOB_10_STEP_51)
      Contact( "Unit1.Em7.ControlNodes".conveyor.sequence.status.seqActive )
      wire#w1
      Coil( "Unit1.Em7.ControlNodes".conveyor."step".action[1051] )
   END_RUNG
   RUNG wire#w1
      Contact( "Unit1.EmNodes".emRelations.em3.monitoring.Jobstatus.WebGuidMotionSemiStepJob6.completed )
      Contact( "Unit1.Em7.ControlNodes".ConveyorEmpty )
      Coil( "Unit1.Em7.ControlNodes".conveyor."step".transition[1051] )
   END_RUNG
   RUNG wire#w1
      Contact( "Unit1.Em7.ControlNodes".conveyor."step".transition[1051] )
      { S7_Templates := "time_type := Time" } #statTonTimer[1051].TON(pt := #SeqDelayTime, et =>)
      wire#w2
      { S7_Templates := "SrcType := Int" } NE_Contact(in1 := "Unit1.EmNodes".emRelations.em6.monitoring.UserDefine.GuageRnRType3PartsCountPV, in2 := "Unit1.EmNodes".emRelations.em6.monitoring.UserDefine.GuageRnRType3PartsCountSV)
      Move(in := #JOB_10_STEP_61, out1 => "Unit1.Em7.ControlNodes".conveyor.sequence.status.nextStep)
   END_RUNG
   RUNG wire#w2
      { S7_Templates := "SrcType := Int" } EQ_Contact(in1 := "Unit1.EmNodes".emRelations.em6.monitoring.UserDefine.GuageRnRType3PartsCountPV, in2 := "Unit1.EmNodes".emRelations.em6.monitoring.UserDefine.GuageRnRType3PartsCountSV)
      Move(in := #JOB_10_STEP_91, out1 => "Unit1.Em7.ControlNodes".conveyor.sequence.status.nextStep)
   END_RUNG
   // the same network as SCL:
   "Unit1.Em7.ControlNodes".conveyor."step".action[1051] := ("Unit1.Em7.ControlNodes".conveyor.sequence.status.currentStep = #JOB_10_STEP_51) AND "Unit1.Em7.ControlNodes".conveyor.sequence.status.seqActive;
   "Unit1.Em7.ControlNodes".conveyor."step".transition[1051] := ("Unit1.Em7.ControlNodes".conveyor.sequence.status.currentStep = #JOB_10_STEP_51) AND "Unit1.Em7.ControlNodes".conveyor.sequence.status.seqActive AND "Unit1.EmNodes".emRelations.em3.monitoring.Jobstatus.WebGuidMotionSemiStepJob6.completed AND "Unit1.Em7.ControlNodes".ConveyorEmpty;
   #statTonTimer[1051].TON(IN := ("Unit1.Em7.ControlNodes".conveyor.sequence.status.currentStep = #JOB_10_STEP_51) AND "Unit1.Em7.ControlNodes".conveyor.sequence.status.seqActive AND "Unit1.Em7.ControlNodes".conveyor."step".transition[1051],
                           PT := #SeqDelayTime);
   IF #statTonTimer[1051].Q AND ("Unit1.EmNodes".emRelations.em6.monitoring.UserDefine.GuageRnRType3PartsCountPV <> "Unit1.EmNodes".emRelations.em6.monitoring.UserDefine.GuageRnRType3PartsCountSV) THEN
       "Unit1.Em7.ControlNodes".conveyor.sequence.status.nextStep := #JOB_10_STEP_61;
   END_IF;
   IF #statTonTimer[1051].Q AND ("Unit1.EmNodes".emRelations.em6.monitoring.UserDefine.GuageRnRType3PartsCountPV = "Unit1.EmNodes".emRelations.em6.monitoring.UserDefine.GuageRnRType3PartsCountSV) THEN
       "Unit1.Em7.ControlNodes".conveyor.sequence.status.nextStep := #JOB_10_STEP_91;
   END_IF;
END_REGION

REGION Network 38: Step[1061] : GaugeRnR3 Loading Request
   RUNG wire#powerrail
      { S7_Templates := "SrcType := DInt" } EQ_Contact(in1 := "Unit1.Em7.ControlNodes".conveyor.sequence.status.currentStep, in2 := #JOB_10_STEP_61)
      Contact( "Unit1.Em7.ControlNodes".conveyor.sequence.status.seqActive )
      wire#w1
      Coil( "Unit1.Em7.ControlNodes".conveyor."step".action[1061] )
   END_RUNG
   RUNG wire#w1
      Contact( "Unit1.EmNodes".emRelations.em5.monitoring.jobStatus.ManualInPutLoadingJob2.active )
      Coil( "Unit1.Em7.ControlNodes".conveyor."step".transition[1061] )
   END_RUNG
   RUNG wire#w1
      Contact( "Unit1.Em7.ControlNodes".conveyor."step".transition[1061] )
      { S7_Templates := "time_type := Time" } #statTonTimer[1061].TON(pt := #SeqDelayTime, et =>)
      Move(in := #JOB_10_STEP_91, out1 => "Unit1.Em7.ControlNodes".conveyor.sequence.status.nextStep)
   END_RUNG
   // the same network as SCL:
   "Unit1.Em7.ControlNodes".conveyor."step".action[1061] := ("Unit1.Em7.ControlNodes".conveyor.sequence.status.currentStep = #JOB_10_STEP_61) AND "Unit1.Em7.ControlNodes".conveyor.sequence.status.seqActive;
   "Unit1.Em7.ControlNodes".conveyor."step".transition[1061] := ("Unit1.Em7.ControlNodes".conveyor.sequence.status.currentStep = #JOB_10_STEP_61) AND "Unit1.Em7.ControlNodes".conveyor.sequence.status.seqActive AND "Unit1.EmNodes".emRelations.em5.monitoring.jobStatus.ManualInPutLoadingJob2.active;
   #statTonTimer[1061].TON(IN := ("Unit1.Em7.ControlNodes".conveyor.sequence.status.currentStep = #JOB_10_STEP_61) AND "Unit1.Em7.ControlNodes".conveyor.sequence.status.seqActive AND "Unit1.Em7.ControlNodes".conveyor."step".transition[1061],
                           PT := #SeqDelayTime);
   IF #statTonTimer[1061].Q THEN
       "Unit1.Em7.ControlNodes".conveyor.sequence.status.nextStep := #JOB_10_STEP_91;
   END_IF;
END_REGION

REGION Network 39: Step[1091] : JOB[10] Step End
   RUNG wire#powerrail
      { S7_Templates := "SrcType := DInt" } EQ_Contact(in1 := "Unit1.Em7.ControlNodes".conveyor.sequence.status.currentStep, in2 := #JOB_10_STEP_91)
      Contact( "Unit1.Em7.ControlNodes".conveyor.sequence.status.seqActive )
      wire#w1
      Coil( "Unit1.Em7.ControlNodes".conveyor."step".action[1091] )
   END_RUNG
   RUNG wire#w1
      Coil( "Unit1.Em7.ControlNodes".conveyor."step".transition[1091] )
   END_RUNG
   RUNG wire#w1
      Contact( "Unit1.Em7.ControlNodes".conveyor."step".transition[1091] )
      { S7_Templates := "time_type := Time" } #statTonTimer[1091].TON(pt := #SeqNoDelayTime, et =>)
      Move(in := #STEP_IDLE, out1 => "Unit1.Em7.ControlNodes".conveyor.sequence.status.nextStep)
   END_RUNG
   // the same network as SCL:
   "Unit1.Em7.ControlNodes".conveyor."step".action[1091] := ("Unit1.Em7.ControlNodes".conveyor.sequence.status.currentStep = #JOB_10_STEP_91) AND "Unit1.Em7.ControlNodes".conveyor.sequence.status.seqActive;
   "Unit1.Em7.ControlNodes".conveyor."step".transition[1091] := ("Unit1.Em7.ControlNodes".conveyor.sequence.status.currentStep = #JOB_10_STEP_91) AND "Unit1.Em7.ControlNodes".conveyor.sequence.status.seqActive;
   #statTonTimer[1091].TON(IN := ("Unit1.Em7.ControlNodes".conveyor.sequence.status.currentStep = #JOB_10_STEP_91) AND "Unit1.Em7.ControlNodes".conveyor.sequence.status.seqActive AND "Unit1.Em7.ControlNodes".conveyor."step".transition[1091],
                           PT := #SeqNoDelayTime);
   IF #statTonTimer[1091].Q THEN
       "Unit1.Em7.ControlNodes".conveyor.sequence.status.nextStep := #STEP_IDLE;
   END_IF;
END_REGION

REGION Network 40: ******************** JOB[11] C/V Full Charge Check CMD ********************
END_REGION

REGION Network 41: Step [1101] : JOB[11] Condition
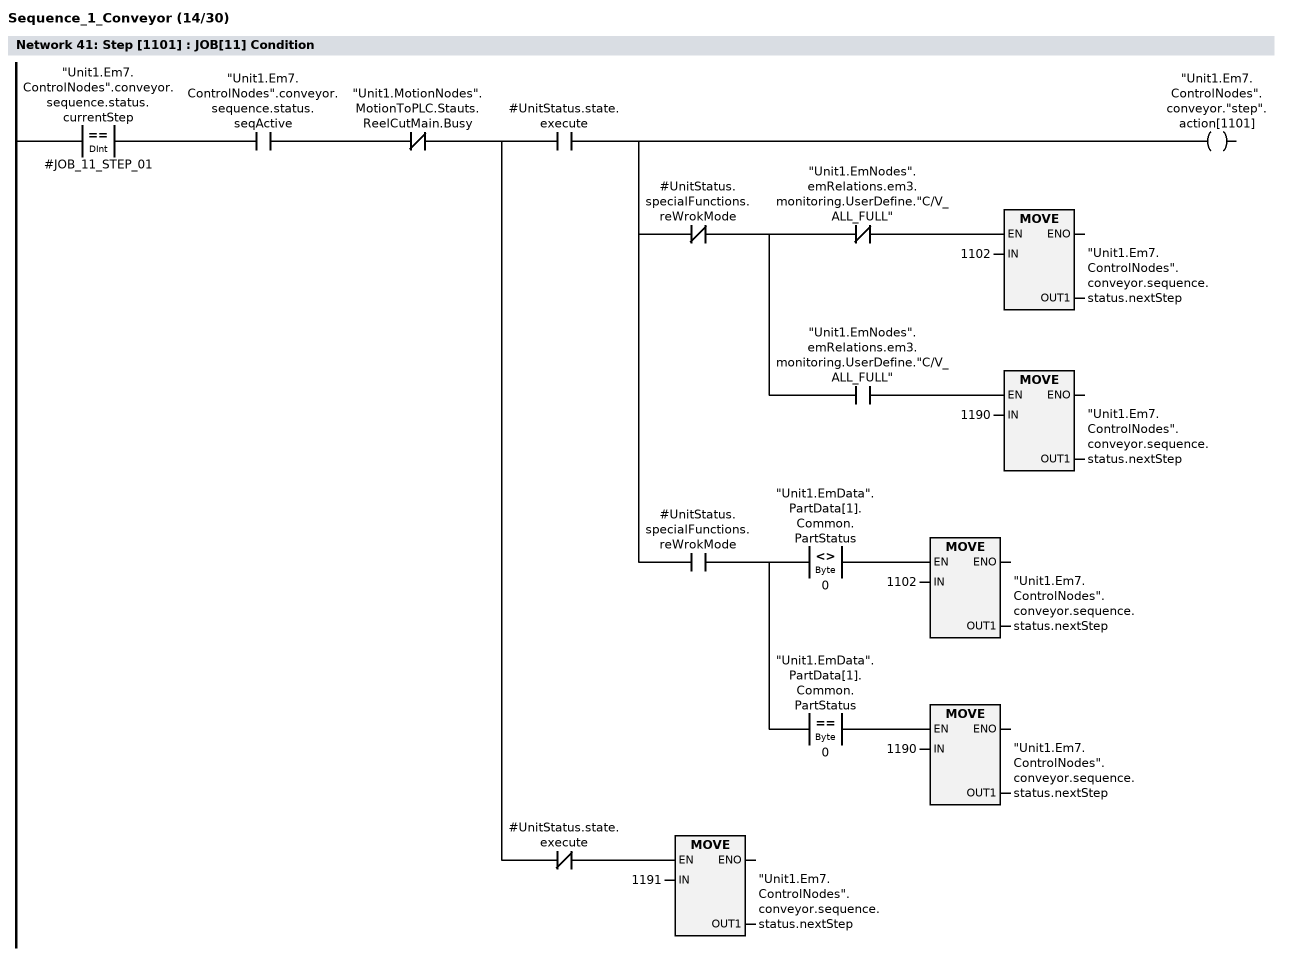
   RUNG wire#powerrail
      { S7_Templates := "SrcType := DInt" } EQ_Contact(in1 := "Unit1.Em7.ControlNodes".conveyor.sequence.status.currentStep, in2 := #JOB_11_STEP_01)
      Contact( "Unit1.Em7.ControlNodes".conveyor.sequence.status.seqActive )
      I_Contact( "Unit1.MotionNodes".MotionToPLC.Stauts.ReelCutMain.Busy )
      wire#w1
      Contact( #UnitStatus.state.execute )
      wire#w2
      Coil( "Unit1.Em7.ControlNodes".conveyor."step".action[1101] )
   END_RUNG
   RUNG wire#w2
      I_Contact( #UnitStatus.specialFunctions.reWrokMode )
      wire#w3
      I_Contact( "Unit1.EmNodes".emRelations.em3.monitoring.UserDefine."C/V_ALL_FULL" )
      Move(in := 1102, out1 => "Unit1.Em7.ControlNodes".conveyor.sequence.status.nextStep)
   END_RUNG
   RUNG wire#w3
      Contact( "Unit1.EmNodes".emRelations.em3.monitoring.UserDefine."C/V_ALL_FULL" )
      Move(in := 1190, out1 => "Unit1.Em7.ControlNodes".conveyor.sequence.status.nextStep)
   END_RUNG
   RUNG wire#w2
      Contact( #UnitStatus.specialFunctions.reWrokMode )
      wire#w4
      { S7_Templates := "SrcType := Byte" } NE_Contact(in1 := "Unit1.EmData".PartData[1].Common.PartStatus, in2 := 0)
      Move(in := 1102, out1 => "Unit1.Em7.ControlNodes".conveyor.sequence.status.nextStep)
   END_RUNG
   RUNG wire#w4
      { S7_Templates := "SrcType := Byte" } EQ_Contact(in1 := "Unit1.EmData".PartData[1].Common.PartStatus, in2 := 0)
      Move(in := 1190, out1 => "Unit1.Em7.ControlNodes".conveyor.sequence.status.nextStep)
   END_RUNG
   RUNG wire#w1
      I_Contact( #UnitStatus.state.execute )
      Move(in := 1191, out1 => "Unit1.Em7.ControlNodes".conveyor.sequence.status.nextStep)
   END_RUNG
   // the same network as SCL:
   #_w1 := ("Unit1.Em7.ControlNodes".conveyor.sequence.status.currentStep = #JOB_11_STEP_01) AND "Unit1.Em7.ControlNodes".conveyor.sequence.status.seqActive AND NOT "Unit1.MotionNodes".MotionToPLC.Stauts.ReelCutMain.Busy;
   "Unit1.Em7.ControlNodes".conveyor."step".action[1101] := #_w1 AND #UnitStatus.state.execute;
   #_w2 := #_w1 AND #UnitStatus.state.execute AND NOT #UnitStatus.specialFunctions.reWrokMode;
   IF #_w2 AND NOT "Unit1.EmNodes".emRelations.em3.monitoring.UserDefine."C/V_ALL_FULL" THEN
       "Unit1.Em7.ControlNodes".conveyor.sequence.status.nextStep := 1102;
   END_IF;
   IF #_w2 AND "Unit1.EmNodes".emRelations.em3.monitoring.UserDefine."C/V_ALL_FULL" THEN
       "Unit1.Em7.ControlNodes".conveyor.sequence.status.nextStep := 1190;
   END_IF;
   #_w3 := #_w1 AND #UnitStatus.state.execute AND #UnitStatus.specialFunctions.reWrokMode;
   IF #_w3 AND ("Unit1.EmData".PartData[1].Common.PartStatus <> 0) THEN
       "Unit1.Em7.ControlNodes".conveyor.sequence.status.nextStep := 1102;
   END_IF;
   IF #_w3 AND ("Unit1.EmData".PartData[1].Common.PartStatus = 0) THEN
       "Unit1.Em7.ControlNodes".conveyor.sequence.status.nextStep := 1190;
   END_IF;
   IF #_w1 AND NOT #UnitStatus.state.execute THEN
       "Unit1.Em7.ControlNodes".conveyor.sequence.status.nextStep := 1191;
   END_IF;
END_REGION

